    CONST robtarget T1339:=[[116.540134,72.670297,13.200015],[0.000000,0.000000,1.000000,0.000000],[0,0,-1,0],[9E+09,9E+09,9E+09,9E+09,9E+09,9E+09]];
    CONST robtarget T1340:=[[116.540134,87.329711,13.200015],[0.000000,0.000000,1.000000,0.000000],[0,0,-1,0],[9E+09,9E+09,9E+09,9E+09,9E+09,9E+09]];
    CONST robtarget T1341:=[[116.540134,114.115099,13.200015],[0.000000,0.000000,1.000000,0.000000],[0,0,-1,0],[9E+09,9E+09,9E+09,9E+09,9E+09,9E+09]];
    CONST robtarget T1342:=[[117.800139,112.721391,13.200015],[0.000000,0.000000,1.000000,0.000000],[0,0,-1,0],[9E+09,9E+09,9E+09,9E+09,9E+09,9E+09]];
    CONST robtarget T1343:=[[117.800139,86.948670,13.200015],[0.000000,0.000000,1.000000,0.000000],[0,0,-1,0],[9E+09,9E+09,9E+09,9E+09,9E+09,9E+09]];
    CONST robtarget T1344:=[[117.800139,73.051337,13.200015],[0.000000,0.000000,1.000000,0.000000],[0,0,-1,0],[9E+09,9E+09,9E+09,9E+09,9E+09,9E+09]];
    CONST robtarget T1345:=[[117.800139,47.278617,13.200015],[0.000000,0.000000,1.000000,0.000000],[0,0,-1,0],[9E+09,9E+09,9E+09,9E+09,9E+09,9E+09]];
    CONST robtarget T1346:=[[119.060143,48.787854,13.200015],[0.000000,0.000000,1.000000,0.000000],[0,0,-1,0],[9E+09,9E+09,9E+09,9E+09,9E+09,9E+09]];
    CONST robtarget T1347:=[[119.060143,73.708792,13.200015],[0.000000,0.000000,1.000000,0.000000],[0,0,-1,0],[9E+09,9E+09,9E+09,9E+09,9E+09,9E+09]];
    CONST robtarget T1348:=[[119.060143,86.291215,13.200015],[0.000000,0.000000,1.000000,0.000000],[0,0,-1,0],[9E+09,9E+09,9E+09,9E+09,9E+09,9E+09]];
    CONST robtarget T1349:=[[119.060143,111.212154,13.200015],[0.000000,0.000000,1.000000,0.000000],[0,0,-1,0],[9E+09,9E+09,9E+09,9E+09,9E+09,9E+09]];
    CONST robtarget T1350:=[[120.320148,109.560940,13.200015],[0.000000,0.000000,1.000000,0.000000],[0,0,-1,0],[9E+09,9E+09,9E+09,9E+09,9E+09,9E+09]];
    CONST robtarget T1351:=[[120.320148,85.271589,13.200015],[0.000000,0.000000,1.000000,0.000000],[0,0,-1,0],[9E+09,9E+09,9E+09,9E+09,9E+09,9E+09]];
    CONST robtarget T1352:=[[120.320148,74.728418,13.200015],[0.000000,0.000000,1.000000,0.000000],[0,0,-1,0],[9E+09,9E+09,9E+09,9E+09,9E+09,9E+09]];
    CONST robtarget T1353:=[[120.320148,50.439068,13.200015],[0.000000,0.000000,1.000000,0.000000],[0,0,-1,0],[9E+09,9E+09,9E+09,9E+09,9E+09,9E+09]];
    CONST robtarget T1354:=[[121.580152,52.240778,13.200015],[0.000000,0.000000,1.000000,0.000000],[0,0,-1,0],[9E+09,9E+09,9E+09,9E+09,9E+09,9E+09]];
    CONST robtarget T1355:=[[121.580152,76.422528,13.200015],[0.000000,0.000000,1.000000,0.000000],[0,0,-1,0],[9E+09,9E+09,9E+09,9E+09,9E+09,9E+09]];
    CONST robtarget T1356:=[[121.580152,83.577479,13.200015],[0.000000,0.000000,1.000000,0.000000],[0,0,-1,0],[9E+09,9E+09,9E+09,9E+09,9E+09,9E+09]];
    CONST robtarget T1357:=[[121.580152,107.759230,13.200015],[0.000000,0.000000,1.000000,0.000000],[0,0,-1,0],[9E+09,9E+09,9E+09,9E+09,9E+09,9E+09]];
    CONST robtarget T1358:=[[122.840157,105.775934,13.200015],[0.000000,0.000000,1.000000,0.000000],[0,0,-1,0],[9E+09,9E+09,9E+09,9E+09,9E+09,9E+09]];
    CONST robtarget T1359:=[[122.840157,54.224074,13.200015],[0.000000,0.000000,1.000000,0.000000],[0,0,-1,0],[9E+09,9E+09,9E+09,9E+09,9E+09,9E+09]];
    CONST robtarget T1360:=[[124.100161,56.444690,13.200015],[0.000000,0.000000,1.000000,0.000000],[0,0,-1,0],[9E+09,9E+09,9E+09,9E+09,9E+09,9E+09]];
    CONST robtarget T1361:=[[124.100161,103.555317,13.200015],[0.000000,0.000000,1.000000,0.000000],[0,0,-1,0],[9E+09,9E+09,9E+09,9E+09,9E+09,9E+09]];
    CONST robtarget T1362:=[[125.360166,101.007928,13.200015],[0.000000,0.000000,1.000000,0.000000],[0,0,-1,0],[9E+09,9E+09,9E+09,9E+09,9E+09,9E+09]];
    CONST robtarget T1363:=[[125.360166,58.992080,13.200015],[0.000000,0.000000,1.000000,0.000000],[0,0,-1,0],[9E+09,9E+09,9E+09,9E+09,9E+09,9E+09]];
    CONST robtarget T1364:=[[126.620170,61.953657,13.200015],[0.000000,0.000000,1.000000,0.000000],[0,0,-1,0],[9E+09,9E+09,9E+09,9E+09,9E+09,9E+09]];
    CONST robtarget T1365:=[[126.620170,98.046351,13.200015],[0.000000,0.000000,1.000000,0.000000],[0,0,-1,0],[9E+09,9E+09,9E+09,9E+09,9E+09,9E+09]];
    CONST robtarget T1366:=[[127.880175,94.360756,13.200015],[0.000000,0.000000,1.000000,0.000000],[0,0,-1,0],[9E+09,9E+09,9E+09,9E+09,9E+09,9E+09]];
    CONST robtarget T1367:=[[127.880175,65.639251,13.200015],[0.000000,0.000000,1.000000,0.000000],[0,0,-1,0],[9E+09,9E+09,9E+09,9E+09,9E+09,9E+09]];
    CONST robtarget T1368:=[[129.140179,70.797151,13.200015],[0.000000,0.000000,1.000000,0.000000],[0,0,-1,0],[9E+09,9E+09,9E+09,9E+09,9E+09,9E+09]];
    CONST robtarget T1369:=[[129.140179,89.202857,13.200015],[0.000000,0.000000,1.000000,0.000000],[0,0,-1,0],[9E+09,9E+09,9E+09,9E+09,9E+09,9E+09]];
    CONST robtarget T1370:=[[129.140179,70.797151,13.900025],[0.000000,0.000000,1.000000,0.000000],[0,0,-1,0],[9E+09,9E+09,9E+09,9E+09,9E+09,9E+09]];
    CONST robtarget T1371:=[[129.140179,89.202857,13.900025],[0.000000,0.000000,1.000000,0.000000],[0,0,-1,0],[9E+09,9E+09,9E+09,9E+09,9E+09,9E+09]];
    CONST robtarget T1372:=[[129.140179,70.797151,13.900025],[0.000000,0.000000,1.000000,0.000000],[0,0,-1,0],[9E+09,9E+09,9E+09,9E+09,9E+09,9E+09]];
    CONST robtarget T1373:=[[129.140179,89.202857,13.900025],[0.000000,0.000000,1.000000,0.000000],[0,0,-1,0],[9E+09,9E+09,9E+09,9E+09,9E+09,9E+09]];
    CONST robtarget T1374:=[[127.880175,94.360756,13.900025],[0.000000,0.000000,1.000000,0.000000],[0,0,-1,0],[9E+09,9E+09,9E+09,9E+09,9E+09,9E+09]];
    CONST robtarget T1375:=[[127.880175,65.639251,13.900025],[0.000000,0.000000,1.000000,0.000000],[0,0,-1,0],[9E+09,9E+09,9E+09,9E+09,9E+09,9E+09]];
    CONST robtarget T1376:=[[126.620170,61.953657,13.900025],[0.000000,0.000000,1.000000,0.000000],[0,0,-1,0],[9E+09,9E+09,9E+09,9E+09,9E+09,9E+09]];
    CONST robtarget T1377:=[[126.620170,98.046351,13.900025],[0.000000,0.000000,1.000000,0.000000],[0,0,-1,0],[9E+09,9E+09,9E+09,9E+09,9E+09,9E+09]];
    CONST robtarget T1378:=[[125.360166,101.007928,13.900025],[0.000000,0.000000,1.000000,0.000000],[0,0,-1,0],[9E+09,9E+09,9E+09,9E+09,9E+09,9E+09]];
    CONST robtarget T1379:=[[125.360166,58.992080,13.900025],[0.000000,0.000000,1.000000,0.000000],[0,0,-1,0],[9E+09,9E+09,9E+09,9E+09,9E+09,9E+09]];
    CONST robtarget T1380:=[[124.100161,56.444690,13.900025],[0.000000,0.000000,1.000000,0.000000],[0,0,-1,0],[9E+09,9E+09,9E+09,9E+09,9E+09,9E+09]];
    CONST robtarget T1381:=[[124.100161,103.555317,13.900025],[0.000000,0.000000,1.000000,0.000000],[0,0,-1,0],[9E+09,9E+09,9E+09,9E+09,9E+09,9E+09]];
    CONST robtarget T1382:=[[122.840157,105.775934,13.900025],[0.000000,0.000000,1.000000,0.000000],[0,0,-1,0],[9E+09,9E+09,9E+09,9E+09,9E+09,9E+09]];
    CONST robtarget T1383:=[[122.840157,54.224074,13.900025],[0.000000,0.000000,1.000000,0.000000],[0,0,-1,0],[9E+09,9E+09,9E+09,9E+09,9E+09,9E+09]];
    CONST robtarget T1384:=[[121.580152,52.240778,13.900025],[0.000000,0.000000,1.000000,0.000000],[0,0,-1,0],[9E+09,9E+09,9E+09,9E+09,9E+09,9E+09]];
    CONST robtarget T1385:=[[121.580152,76.422528,13.900025],[0.000000,0.000000,1.000000,0.000000],[0,0,-1,0],[9E+09,9E+09,9E+09,9E+09,9E+09,9E+09]];
    CONST robtarget T1386:=[[121.580152,83.577479,13.900025],[0.000000,0.000000,1.000000,0.000000],[0,0,-1,0],[9E+09,9E+09,9E+09,9E+09,9E+09,9E+09]];
    CONST robtarget T1387:=[[121.580152,107.759230,13.900025],[0.000000,0.000000,1.000000,0.000000],[0,0,-1,0],[9E+09,9E+09,9E+09,9E+09,9E+09,9E+09]];
    CONST robtarget T1388:=[[120.320148,109.560940,13.900025],[0.000000,0.000000,1.000000,0.000000],[0,0,-1,0],[9E+09,9E+09,9E+09,9E+09,9E+09,9E+09]];
    CONST robtarget T1389:=[[120.320148,85.271589,13.900025],[0.000000,0.000000,1.000000,0.000000],[0,0,-1,0],[9E+09,9E+09,9E+09,9E+09,9E+09,9E+09]];
    CONST robtarget T1390:=[[120.320148,74.728418,13.900025],[0.000000,0.000000,1.000000,0.000000],[0,0,-1,0],[9E+09,9E+09,9E+09,9E+09,9E+09,9E+09]];
    CONST robtarget T1391:=[[120.320148,50.439068,13.900025],[0.000000,0.000000,1.000000,0.000000],[0,0,-1,0],[9E+09,9E+09,9E+09,9E+09,9E+09,9E+09]];
    CONST robtarget T1392:=[[119.060143,48.787854,13.900025],[0.000000,0.000000,1.000000,0.000000],[0,0,-1,0],[9E+09,9E+09,9E+09,9E+09,9E+09,9E+09]];
    CONST robtarget T1393:=[[119.060143,73.708792,13.900025],[0.000000,0.000000,1.000000,0.000000],[0,0,-1,0],[9E+09,9E+09,9E+09,9E+09,9E+09,9E+09]];
    CONST robtarget T1394:=[[119.060143,86.291215,13.900025],[0.000000,0.000000,1.000000,0.000000],[0,0,-1,0],[9E+09,9E+09,9E+09,9E+09,9E+09,9E+09]];
    CONST robtarget T1395:=[[119.060143,111.212154,13.900025],[0.000000,0.000000,1.000000,0.000000],[0,0,-1,0],[9E+09,9E+09,9E+09,9E+09,9E+09,9E+09]];
    CONST robtarget T1396:=[[117.800139,112.721391,13.900025],[0.000000,0.000000,1.000000,0.000000],[0,0,-1,0],[9E+09,9E+09,9E+09,9E+09,9E+09,9E+09]];
    CONST robtarget T1397:=[[117.800139,86.948670,13.900025],[0.000000,0.000000,1.000000,0.000000],[0,0,-1,0],[9E+09,9E+09,9E+09,9E+09,9E+09,9E+09]];
    CONST robtarget T1398:=[[117.800139,73.051337,13.900025],[0.000000,0.000000,1.000000,0.000000],[0,0,-1,0],[9E+09,9E+09,9E+09,9E+09,9E+09,9E+09]];
    CONST robtarget T1399:=[[117.800139,47.278617,13.900025],[0.000000,0.000000,1.000000,0.000000],[0,0,-1,0],[9E+09,9E+09,9E+09,9E+09,9E+09,9E+09]];
    CONST robtarget T1400:=[[116.540134,45.884908,13.900025],[0.000000,0.000000,1.000000,0.000000],[0,0,-1,0],[9E+09,9E+09,9E+09,9E+09,9E+09,9E+09]];
    CONST robtarget T1401:=[[116.540134,72.670297,13.900025],[0.000000,0.000000,1.000000,0.000000],[0,0,-1,0],[9E+09,9E+09,9E+09,9E+09,9E+09,9E+09]];
    CONST robtarget T1402:=[[116.540134,87.329711,13.900025],[0.000000,0.000000,1.000000,0.000000],[0,0,-1,0],[9E+09,9E+09,9E+09,9E+09,9E+09,9E+09]];
    CONST robtarget T1403:=[[116.540134,114.115099,13.900025],[0.000000,0.000000,1.000000,0.000000],[0,0,-1,0],[9E+09,9E+09,9E+09,9E+09,9E+09,9E+09]];
    CONST robtarget T1404:=[[115.280130,115.412758,13.900025],[0.000000,0.000000,1.000000,0.000000],[0,0,-1,0],[9E+09,9E+09,9E+09,9E+09,9E+09,9E+09]];
    CONST robtarget T1405:=[[115.280130,87.487316,13.900025],[0.000000,0.000000,1.000000,0.000000],[0,0,-1,0],[9E+09,9E+09,9E+09,9E+09,9E+09,9E+09]];
    CONST robtarget T1406:=[[115.280130,72.512692,13.900025],[0.000000,0.000000,1.000000,0.000000],[0,0,-1,0],[9E+09,9E+09,9E+09,9E+09,9E+09,9E+09]];
    CONST robtarget T1407:=[[115.280130,44.587250,13.900025],[0.000000,0.000000,1.000000,0.000000],[0,0,-1,0],[9E+09,9E+09,9E+09,9E+09,9E+09,9E+09]];
    CONST robtarget T1408:=[[114.020125,43.373063,13.900025],[0.000000,0.000000,1.000000,0.000000],[0,0,-1,0],[9E+09,9E+09,9E+09,9E+09,9E+09,9E+09]];
    CONST robtarget T1409:=[[114.020125,72.576253,13.900025],[0.000000,0.000000,1.000000,0.000000],[0,0,-1,0],[9E+09,9E+09,9E+09,9E+09,9E+09,9E+09]];
    CONST robtarget T1410:=[[114.020125,87.423755,13.900025],[0.000000,0.000000,1.000000,0.000000],[0,0,-1,0],[9E+09,9E+09,9E+09,9E+09,9E+09,9E+09]];
    CONST robtarget T1411:=[[114.020125,116.626944,13.900025],[0.000000,0.000000,1.000000,0.000000],[0,0,-1,0],[9E+09,9E+09,9E+09,9E+09,9E+09,9E+09]];
    CONST robtarget T1412:=[[112.760121,117.767805,13.900025],[0.000000,0.000000,1.000000,0.000000],[0,0,-1,0],[9E+09,9E+09,9E+09,9E+09,9E+09,9E+09]];
    CONST robtarget T1413:=[[112.760121,87.152583,13.900025],[0.000000,0.000000,1.000000,0.000000],[0,0,-1,0],[9E+09,9E+09,9E+09,9E+09,9E+09,9E+09]];
    CONST robtarget T1414:=[[112.760121,72.847425,13.900025],[0.000000,0.000000,1.000000,0.000000],[0,0,-1,0],[9E+09,9E+09,9E+09,9E+09,9E+09,9E+09]];
    CONST robtarget T1415:=[[112.760121,42.232203,13.900025],[0.000000,0.000000,1.000000,0.000000],[0,0,-1,0],[9E+09,9E+09,9E+09,9E+09,9E+09,9E+09]];
    CONST robtarget T1416:=[[111.500116,41.180273,13.900025],[0.000000,0.000000,1.000000,0.000000],[0,0,-1,0],[9E+09,9E+09,9E+09,9E+09,9E+09,9E+09]];
    CONST robtarget T1417:=[[111.500116,73.379202,13.900025],[0.000000,0.000000,1.000000,0.000000],[0,0,-1,0],[9E+09,9E+09,9E+09,9E+09,9E+09,9E+09]];
    CONST robtarget T1418:=[[111.500116,86.620805,13.900025],[0.000000,0.000000,1.000000,0.000000],[0,0,-1,0],[9E+09,9E+09,9E+09,9E+09,9E+09,9E+09]];
    CONST robtarget T1419:=[[111.500116,118.819735,13.900025],[0.000000,0.000000,1.000000,0.000000],[0,0,-1,0],[9E+09,9E+09,9E+09,9E+09,9E+09,9E+09]];
    CONST robtarget T1420:=[[110.240112,119.803025,13.900025],[0.000000,0.000000,1.000000,0.000000],[0,0,-1,0],[9E+09,9E+09,9E+09,9E+09,9E+09,9E+09]];
    CONST robtarget T1421:=[[110.240112,85.779969,13.900025],[0.000000,0.000000,1.000000,0.000000],[0,0,-1,0],[9E+09,9E+09,9E+09,9E+09,9E+09,9E+09]];
    CONST robtarget T1422:=[[110.240112,74.220038,13.900025],[0.000000,0.000000,1.000000,0.000000],[0,0,-1,0],[9E+09,9E+09,9E+09,9E+09,9E+09,9E+09]];
    CONST robtarget T1423:=[[110.240112,40.196983,13.900025],[0.000000,0.000000,1.000000,0.000000],[0,0,-1,0],[9E+09,9E+09,9E+09,9E+09,9E+09,9E+09]];
    CONST robtarget T1424:=[[108.980107,39.265681,13.900025],[0.000000,0.000000,1.000000,0.000000],[0,0,-1,0],[9E+09,9E+09,9E+09,9E+09,9E+09,9E+09]];
    CONST robtarget T1425:=[[108.980107,75.547902,13.900025],[0.000000,0.000000,1.000000,0.000000],[0,0,-1,0],[9E+09,9E+09,9E+09,9E+09,9E+09,9E+09]];
    CONST robtarget T1426:=[[108.980107,84.452106,13.900025],[0.000000,0.000000,1.000000,0.000000],[0,0,-1,0],[9E+09,9E+09,9E+09,9E+09,9E+09,9E+09]];
    CONST robtarget T1427:=[[108.980107,120.734326,13.900025],[0.000000,0.000000,1.000000,0.000000],[0,0,-1,0],[9E+09,9E+09,9E+09,9E+09,9E+09,9E+09]];
    CONST robtarget T1428:=[[107.720103,121.607260,13.900025],[0.000000,0.000000,1.000000,0.000000],[0,0,-1,0],[9E+09,9E+09,9E+09,9E+09,9E+09,9E+09]];
    CONST robtarget T1429:=[[107.720103,81.789524,13.900025],[0.000000,0.000000,1.000000,0.000000],[0,0,-1,0],[9E+09,9E+09,9E+09,9E+09,9E+09,9E+09]];
    CONST robtarget T1430:=[[107.720103,78.210483,13.900025],[0.000000,0.000000,1.000000,0.000000],[0,0,-1,0],[9E+09,9E+09,9E+09,9E+09,9E+09,9E+09]];
    CONST robtarget T1431:=[[107.720103,38.392748,13.900025],[0.000000,0.000000,1.000000,0.000000],[0,0,-1,0],[9E+09,9E+09,9E+09,9E+09,9E+09,9E+09]];
    CONST robtarget T1432:=[[106.460098,37.589739,13.900025],[0.000000,0.000000,1.000000,0.000000],[0,0,-1,0],[9E+09,9E+09,9E+09,9E+09,9E+09,9E+09]];
    CONST robtarget T1433:=[[106.460098,122.410268,13.900025],[0.000000,0.000000,1.000000,0.000000],[0,0,-1,0],[9E+09,9E+09,9E+09,9E+09,9E+09,9E+09]];
    CONST robtarget T1434:=[[105.200094,123.174878,13.900025],[0.000000,0.000000,1.000000,0.000000],[0,0,-1,0],[9E+09,9E+09,9E+09,9E+09,9E+09,9E+09]];
    CONST robtarget T1435:=[[105.200094,36.825129,13.900025],[0.000000,0.000000,1.000000,0.000000],[0,0,-1,0],[9E+09,9E+09,9E+09,9E+09,9E+09,9E+09]];
    CONST robtarget T1436:=[[103.940089,36.110177,13.900025],[0.000000,0.000000,1.000000,0.000000],[0,0,-1,0],[9E+09,9E+09,9E+09,9E+09,9E+09,9E+09]];
    CONST robtarget T1437:=[[103.940089,123.889831,13.900025],[0.000000,0.000000,1.000000,0.000000],[0,0,-1,0],[9E+09,9E+09,9E+09,9E+09,9E+09,9E+09]];
    CONST robtarget T1438:=[[102.680085,124.546114,13.900025],[0.000000,0.000000,1.000000,0.000000],[0,0,-1,0],[9E+09,9E+09,9E+09,9E+09,9E+09,9E+09]];
    CONST robtarget T1439:=[[102.680085,35.453894,13.900025],[0.000000,0.000000,1.000000,0.000000],[0,0,-1,0],[9E+09,9E+09,9E+09,9E+09,9E+09,9E+09]];
    CONST robtarget T1440:=[[101.420080,34.827050,13.900025],[0.000000,0.000000,1.000000,0.000000],[0,0,-1,0],[9E+09,9E+09,9E+09,9E+09,9E+09,9E+09]];
    CONST robtarget T1441:=[[101.420080,125.172958,13.900025],[0.000000,0.000000,1.000000,0.000000],[0,0,-1,0],[9E+09,9E+09,9E+09,9E+09,9E+09,9E+09]];
    CONST robtarget T1442:=[[100.160076,125.745278,13.900025],[0.000000,0.000000,1.000000,0.000000],[0,0,-1,0],[9E+09,9E+09,9E+09,9E+09,9E+09,9E+09]];
    CONST robtarget T1443:=[[100.160076,34.254730,13.900025],[0.000000,0.000000,1.000000,0.000000],[0,0,-1,0],[9E+09,9E+09,9E+09,9E+09,9E+09,9E+09]];
    CONST robtarget T1444:=[[98.900071,33.722290,13.900025],[0.000000,0.000000,1.000000,0.000000],[0,0,-1,0],[9E+09,9E+09,9E+09,9E+09,9E+09,9E+09]];
    CONST robtarget T1445:=[[98.900071,126.277717,13.900025],[0.000000,0.000000,1.000000,0.000000],[0,0,-1,0],[9E+09,9E+09,9E+09,9E+09,9E+09,9E+09]];
    CONST robtarget T1446:=[[97.640067,126.783143,13.900025],[0.000000,0.000000,1.000000,0.000000],[0,0,-1,0],[9E+09,9E+09,9E+09,9E+09,9E+09,9E+09]];
    CONST robtarget T1447:=[[97.640067,33.216864,13.900025],[0.000000,0.000000,1.000000,0.000000],[0,0,-1,0],[9E+09,9E+09,9E+09,9E+09,9E+09,9E+09]];
    CONST robtarget T1448:=[[96.380062,32.772318,13.900025],[0.000000,0.000000,1.000000,0.000000],[0,0,-1,0],[9E+09,9E+09,9E+09,9E+09,9E+09,9E+09]];
    CONST robtarget T1449:=[[96.380062,127.227690,13.900025],[0.000000,0.000000,1.000000,0.000000],[0,0,-1,0],[9E+09,9E+09,9E+09,9E+09,9E+09,9E+09]];
    CONST robtarget T1450:=[[95.120058,127.652167,13.900025],[0.000000,0.000000,1.000000,0.000000],[0,0,-1,0],[9E+09,9E+09,9E+09,9E+09,9E+09,9E+09]];
    CONST robtarget T1451:=[[95.120058,32.347841,13.900025],[0.000000,0.000000,1.000000,0.000000],[0,0,-1,0],[9E+09,9E+09,9E+09,9E+09,9E+09,9E+09]];
    CONST robtarget T1452:=[[93.860053,31.969479,13.900025],[0.000000,0.000000,1.000000,0.000000],[0,0,-1,0],[9E+09,9E+09,9E+09,9E+09,9E+09,9E+09]];
    CONST robtarget T1453:=[[93.860053,128.030529,13.900025],[0.000000,0.000000,1.000000,0.000000],[0,0,-1,0],[9E+09,9E+09,9E+09,9E+09,9E+09,9E+09]];
    CONST robtarget T1454:=[[92.600049,128.374988,13.900025],[0.000000,0.000000,1.000000,0.000000],[0,0,-1,0],[9E+09,9E+09,9E+09,9E+09,9E+09,9E+09]];
    CONST robtarget T1455:=[[92.600049,31.625019,13.900025],[0.000000,0.000000,1.000000,0.000000],[0,0,-1,0],[9E+09,9E+09,9E+09,9E+09,9E+09,9E+09]];
    CONST robtarget T1456:=[[91.340044,31.307526,13.900025],[0.000000,0.000000,1.000000,0.000000],[0,0,-1,0],[9E+09,9E+09,9E+09,9E+09,9E+09,9E+09]];
    CONST robtarget T1457:=[[91.340044,128.692481,13.900025],[0.000000,0.000000,1.000000,0.000000],[0,0,-1,0],[9E+09,9E+09,9E+09,9E+09,9E+09,9E+09]];
    CONST robtarget T1458:=[[90.080040,128.960575,13.900025],[0.000000,0.000000,1.000000,0.000000],[0,0,-1,0],[9E+09,9E+09,9E+09,9E+09,9E+09,9E+09]];
    CONST robtarget T1459:=[[90.080040,31.039433,13.900025],[0.000000,0.000000,1.000000,0.000000],[0,0,-1,0],[9E+09,9E+09,9E+09,9E+09,9E+09,9E+09]];
    CONST robtarget T1460:=[[88.820035,30.786444,13.900025],[0.000000,0.000000,1.000000,0.000000],[0,0,-1,0],[9E+09,9E+09,9E+09,9E+09,9E+09,9E+09]];
    CONST robtarget T1461:=[[88.820035,129.213563,13.900025],[0.000000,0.000000,1.000000,0.000000],[0,0,-1,0],[9E+09,9E+09,9E+09,9E+09,9E+09,9E+09]];
    CONST robtarget T1462:=[[87.560031,129.413129,13.900025],[0.000000,0.000000,1.000000,0.000000],[0,0,-1,0],[9E+09,9E+09,9E+09,9E+09,9E+09,9E+09]];
    CONST robtarget T1463:=[[87.560031,30.586879,13.900025],[0.000000,0.000000,1.000000,0.000000],[0,0,-1,0],[9E+09,9E+09,9E+09,9E+09,9E+09,9E+09]];
    CONST robtarget T1464:=[[86.300026,30.406130,13.900025],[0.000000,0.000000,1.000000,0.000000],[0,0,-1,0],[9E+09,9E+09,9E+09,9E+09,9E+09,9E+09]];
    CONST robtarget T1465:=[[86.300026,40.937335,13.900025],[0.000000,0.000000,1.000000,0.000000],[0,0,-1,0],[9E+09,9E+09,9E+09,9E+09,9E+09,9E+09]];
    CONST robtarget T1466:=[[86.300026,49.062665,13.900025],[0.000000,0.000000,1.000000,0.000000],[0,0,-1,0],[9E+09,9E+09,9E+09,9E+09,9E+09,9E+09]];
    CONST robtarget T1467:=[[86.300026,75.937339,13.900025],[0.000000,0.000000,1.000000,0.000000],[0,0,-1,0],[9E+09,9E+09,9E+09,9E+09,9E+09,9E+09]];
    CONST robtarget T1468:=[[86.300026,84.062668,13.900025],[0.000000,0.000000,1.000000,0.000000],[0,0,-1,0],[9E+09,9E+09,9E+09,9E+09,9E+09,9E+09]];
    CONST robtarget T1469:=[[86.300026,110.937342,13.900025],[0.000000,0.000000,1.000000,0.000000],[0,0,-1,0],[9E+09,9E+09,9E+09,9E+09,9E+09,9E+09]];
    CONST robtarget T1470:=[[86.300026,119.062672,13.900025],[0.000000,0.000000,1.000000,0.000000],[0,0,-1,0],[9E+09,9E+09,9E+09,9E+09,9E+09,9E+09]];
    CONST robtarget T1471:=[[86.300026,129.593877,13.900025],[0.000000,0.000000,1.000000,0.000000],[0,0,-1,0],[9E+09,9E+09,9E+09,9E+09,9E+09,9E+09]];
    CONST robtarget T1472:=[[85.040022,129.735844,13.900025],[0.000000,0.000000,1.000000,0.000000],[0,0,-1,0],[9E+09,9E+09,9E+09,9E+09,9E+09,9E+09]];
    CONST robtarget T1473:=[[85.040022,120.544921,13.900025],[0.000000,0.000000,1.000000,0.000000],[0,0,-1,0],[9E+09,9E+09,9E+09,9E+09,9E+09,9E+09]];
    CONST robtarget T1474:=[[85.040022,109.455091,13.900025],[0.000000,0.000000,1.000000,0.000000],[0,0,-1,0],[9E+09,9E+09,9E+09,9E+09,9E+09,9E+09]];
    CONST robtarget T1475:=[[85.040022,85.544918,13.900025],[0.000000,0.000000,1.000000,0.000000],[0,0,-1,0],[9E+09,9E+09,9E+09,9E+09,9E+09,9E+09]];
    CONST robtarget T1476:=[[85.040022,74.455090,13.900025],[0.000000,0.000000,1.000000,0.000000],[0,0,-1,0],[9E+09,9E+09,9E+09,9E+09,9E+09,9E+09]];
    CONST robtarget T1477:=[[85.040022,50.544916,13.900025],[0.000000,0.000000,1.000000,0.000000],[0,0,-1,0],[9E+09,9E+09,9E+09,9E+09,9E+09,9E+09]];
    CONST robtarget T1478:=[[85.040022,39.455086,13.900025],[0.000000,0.000000,1.000000,0.000000],[0,0,-1,0],[9E+09,9E+09,9E+09,9E+09,9E+09,9E+09]];
    CONST robtarget T1479:=[[85.040022,30.264163,13.900025],[0.000000,0.000000,1.000000,0.000000],[0,0,-1,0],[9E+09,9E+09,9E+09,9E+09,9E+09,9E+09]];
    CONST robtarget T1480:=[[83.780017,30.153959,13.900025],[0.000000,0.000000,1.000000,0.000000],[0,0,-1,0],[9E+09,9E+09,9E+09,9E+09,9E+09,9E+09]];
    CONST robtarget T1481:=[[83.780017,38.524551,13.900025],[0.000000,0.000000,1.000000,0.000000],[0,0,-1,0],[9E+09,9E+09,9E+09,9E+09,9E+09,9E+09]];
    CONST robtarget T1482:=[[83.780017,51.475451,13.900025],[0.000000,0.000000,1.000000,0.000000],[0,0,-1,0],[9E+09,9E+09,9E+09,9E+09,9E+09,9E+09]];
    CONST robtarget T1483:=[[83.780017,73.524553,13.900025],[0.000000,0.000000,1.000000,0.000000],[0,0,-1,0],[9E+09,9E+09,9E+09,9E+09,9E+09,9E+09]];
    CONST robtarget T1484:=[[83.780017,86.475455,13.900025],[0.000000,0.000000,1.000000,0.000000],[0,0,-1,0],[9E+09,9E+09,9E+09,9E+09,9E+09,9E+09]];
    CONST robtarget T1485:=[[83.780017,108.524556,13.900025],[0.000000,0.000000,1.000000,0.000000],[0,0,-1,0],[9E+09,9E+09,9E+09,9E+09,9E+09,9E+09]];
    CONST robtarget T1486:=[[83.780017,121.475457,13.900025],[0.000000,0.000000,1.000000,0.000000],[0,0,-1,0],[9E+09,9E+09,9E+09,9E+09,9E+09,9E+09]];
    CONST robtarget T1487:=[[83.780017,129.846049,13.900025],[0.000000,0.000000,1.000000,0.000000],[0,0,-1,0],[9E+09,9E+09,9E+09,9E+09,9E+09,9E+09]];
    CONST robtarget T1488:=[[82.520013,129.931001,13.900025],[0.000000,0.000000,1.000000,0.000000],[0,0,-1,0],[9E+09,9E+09,9E+09,9E+09,9E+09,9E+09]];
    CONST robtarget T1489:=[[82.520013,122.050628,13.900025],[0.000000,0.000000,1.000000,0.000000],[0,0,-1,0],[9E+09,9E+09,9E+09,9E+09,9E+09,9E+09]];
    CONST robtarget T1490:=[[82.520013,107.949384,13.900025],[0.000000,0.000000,1.000000,0.000000],[0,0,-1,0],[9E+09,9E+09,9E+09,9E+09,9E+09,9E+09]];
    CONST robtarget T1491:=[[82.520013,87.050626,13.900025],[0.000000,0.000000,1.000000,0.000000],[0,0,-1,0],[9E+09,9E+09,9E+09,9E+09,9E+09,9E+09]];
    CONST robtarget T1492:=[[82.520013,72.949381,13.900025],[0.000000,0.000000,1.000000,0.000000],[0,0,-1,0],[9E+09,9E+09,9E+09,9E+09,9E+09,9E+09]];
    CONST robtarget T1493:=[[82.520013,52.050624,13.900025],[0.000000,0.000000,1.000000,0.000000],[0,0,-1,0],[9E+09,9E+09,9E+09,9E+09,9E+09,9E+09]];
    CONST robtarget T1494:=[[82.520013,37.949379,13.900025],[0.000000,0.000000,1.000000,0.000000],[0,0,-1,0],[9E+09,9E+09,9E+09,9E+09,9E+09,9E+09]];
    CONST robtarget T1495:=[[82.520013,30.069007,13.900025],[0.000000,0.000000,1.000000,0.000000],[0,0,-1,0],[9E+09,9E+09,9E+09,9E+09,9E+09,9E+09]];
    CONST robtarget T1496:=[[81.260008,30.028279,13.900025],[0.000000,0.000000,1.000000,0.000000],[0,0,-1,0],[9E+09,9E+09,9E+09,9E+09,9E+09,9E+09]];
    CONST robtarget T1497:=[[81.260008,37.608991,13.900025],[0.000000,0.000000,1.000000,0.000000],[0,0,-1,0],[9E+09,9E+09,9E+09,9E+09,9E+09,9E+09]];
    CONST robtarget T1498:=[[81.260008,52.391011,13.900025],[0.000000,0.000000,1.000000,0.000000],[0,0,-1,0],[9E+09,9E+09,9E+09,9E+09,9E+09,9E+09]];
    CONST robtarget T1499:=[[81.260008,72.608994,13.900025],[0.000000,0.000000,1.000000,0.000000],[0,0,-1,0],[9E+09,9E+09,9E+09,9E+09,9E+09,9E+09]];
    CONST robtarget T1500:=[[81.260008,87.391014,13.900025],[0.000000,0.000000,1.000000,0.000000],[0,0,-1,0],[9E+09,9E+09,9E+09,9E+09,9E+09,9E+09]];
    CONST robtarget T1501:=[[81.260008,107.608996,13.900025],[0.000000,0.000000,1.000000,0.000000],[0,0,-1,0],[9E+09,9E+09,9E+09,9E+09,9E+09,9E+09]];
    CONST robtarget T1502:=[[81.260008,122.391017,13.900025],[0.000000,0.000000,1.000000,0.000000],[0,0,-1,0],[9E+09,9E+09,9E+09,9E+09,9E+09,9E+09]];
    CONST robtarget T1503:=[[81.260008,129.971729,13.900025],[0.000000,0.000000,1.000000,0.000000],[0,0,-1,0],[9E+09,9E+09,9E+09,9E+09,9E+09,9E+09]];
    CONST robtarget T1504:=[[80.000004,130.000008,13.900025],[0.000000,0.000000,1.000000,0.000000],[0,0,-1,0],[9E+09,9E+09,9E+09,9E+09,9E+09,9E+09]];
    CONST robtarget T1505:=[[80.000004,122.487319,13.900025],[0.000000,0.000000,1.000000,0.000000],[0,0,-1,0],[9E+09,9E+09,9E+09,9E+09,9E+09,9E+09]];
    CONST robtarget T1506:=[[80.000004,107.512696,13.900025],[0.000000,0.000000,1.000000,0.000000],[0,0,-1,0],[9E+09,9E+09,9E+09,9E+09,9E+09,9E+09]];
    CONST robtarget T1507:=[[80.000004,87.487316,13.900025],[0.000000,0.000000,1.000000,0.000000],[0,0,-1,0],[9E+09,9E+09,9E+09,9E+09,9E+09,9E+09]];
    CONST robtarget T1508:=[[80.000004,72.512692,13.900025],[0.000000,0.000000,1.000000,0.000000],[0,0,-1,0],[9E+09,9E+09,9E+09,9E+09,9E+09,9E+09]];
    CONST robtarget T1509:=[[80.000004,52.487312,13.900025],[0.000000,0.000000,1.000000,0.000000],[0,0,-1,0],[9E+09,9E+09,9E+09,9E+09,9E+09,9E+09]];
    CONST robtarget T1510:=[[80.000004,37.512688,13.900025],[0.000000,0.000000,1.000000,0.000000],[0,0,-1,0],[9E+09,9E+09,9E+09,9E+09,9E+09,9E+09]];
    CONST robtarget T1511:=[[80.000004,30.000000,13.900025],[0.000000,0.000000,1.000000,0.000000],[0,0,-1,0],[9E+09,9E+09,9E+09,9E+09,9E+09,9E+09]];
    CONST robtarget T1512:=[[78.739999,30.028279,13.900025],[0.000000,0.000000,1.000000,0.000000],[0,0,-1,0],[9E+09,9E+09,9E+09,9E+09,9E+09,9E+09]];
    CONST robtarget T1513:=[[78.739999,37.608991,13.900025],[0.000000,0.000000,1.000000,0.000000],[0,0,-1,0],[9E+09,9E+09,9E+09,9E+09,9E+09,9E+09]];
    CONST robtarget T1514:=[[78.739999,52.391011,13.900025],[0.000000,0.000000,1.000000,0.000000],[0,0,-1,0],[9E+09,9E+09,9E+09,9E+09,9E+09,9E+09]];
    CONST robtarget T1515:=[[78.739999,72.608994,13.900025],[0.000000,0.000000,1.000000,0.000000],[0,0,-1,0],[9E+09,9E+09,9E+09,9E+09,9E+09,9E+09]];
    CONST robtarget T1516:=[[78.739999,87.391014,13.900025],[0.000000,0.000000,1.000000,0.000000],[0,0,-1,0],[9E+09,9E+09,9E+09,9E+09,9E+09,9E+09]];
    CONST robtarget T1517:=[[78.739999,107.608996,13.900025],[0.000000,0.000000,1.000000,0.000000],[0,0,-1,0],[9E+09,9E+09,9E+09,9E+09,9E+09,9E+09]];
    CONST robtarget T1518:=[[78.739999,122.391017,13.900025],[0.000000,0.000000,1.000000,0.000000],[0,0,-1,0],[9E+09,9E+09,9E+09,9E+09,9E+09,9E+09]];
    CONST robtarget T1519:=[[78.739999,129.971729,13.900025],[0.000000,0.000000,1.000000,0.000000],[0,0,-1,0],[9E+09,9E+09,9E+09,9E+09,9E+09,9E+09]];
    CONST robtarget T1520:=[[77.479995,129.931001,13.900025],[0.000000,0.000000,1.000000,0.000000],[0,0,-1,0],[9E+09,9E+09,9E+09,9E+09,9E+09,9E+09]];
    CONST robtarget T1521:=[[77.479995,122.050628,13.900025],[0.000000,0.000000,1.000000,0.000000],[0,0,-1,0],[9E+09,9E+09,9E+09,9E+09,9E+09,9E+09]];
    CONST robtarget T1522:=[[77.479995,107.949384,13.900025],[0.000000,0.000000,1.000000,0.000000],[0,0,-1,0],[9E+09,9E+09,9E+09,9E+09,9E+09,9E+09]];
    CONST robtarget T1523:=[[77.479995,87.050626,13.900025],[0.000000,0.000000,1.000000,0.000000],[0,0,-1,0],[9E+09,9E+09,9E+09,9E+09,9E+09,9E+09]];
    CONST robtarget T1524:=[[77.479995,72.949381,13.900025],[0.000000,0.000000,1.000000,0.000000],[0,0,-1,0],[9E+09,9E+09,9E+09,9E+09,9E+09,9E+09]];
    CONST robtarget T1525:=[[77.479995,52.050624,13.900025],[0.000000,0.000000,1.000000,0.000000],[0,0,-1,0],[9E+09,9E+09,9E+09,9E+09,9E+09,9E+09]];
    CONST robtarget T1526:=[[77.479995,37.949379,13.900025],[0.000000,0.000000,1.000000,0.000000],[0,0,-1,0],[9E+09,9E+09,9E+09,9E+09,9E+09,9E+09]];
    CONST robtarget T1527:=[[77.479995,30.069007,13.900025],[0.000000,0.000000,1.000000,0.000000],[0,0,-1,0],[9E+09,9E+09,9E+09,9E+09,9E+09,9E+09]];
    CONST robtarget T1528:=[[76.219990,30.153959,13.900025],[0.000000,0.000000,1.000000,0.000000],[0,0,-1,0],[9E+09,9E+09,9E+09,9E+09,9E+09,9E+09]];
    CONST robtarget T1529:=[[76.219990,38.524551,13.900025],[0.000000,0.000000,1.000000,0.000000],[0,0,-1,0],[9E+09,9E+09,9E+09,9E+09,9E+09,9E+09]];
    CONST robtarget T1530:=[[76.219990,51.475451,13.900025],[0.000000,0.000000,1.000000,0.000000],[0,0,-1,0],[9E+09,9E+09,9E+09,9E+09,9E+09,9E+09]];
    CONST robtarget T1531:=[[76.219990,73.524553,13.900025],[0.000000,0.000000,1.000000,0.000000],[0,0,-1,0],[9E+09,9E+09,9E+09,9E+09,9E+09,9E+09]];
    CONST robtarget T1532:=[[76.219990,86.475455,13.900025],[0.000000,0.000000,1.000000,0.000000],[0,0,-1,0],[9E+09,9E+09,9E+09,9E+09,9E+09,9E+09]];
    CONST robtarget T1533:=[[76.219990,108.524556,13.900025],[0.000000,0.000000,1.000000,0.000000],[0,0,-1,0],[9E+09,9E+09,9E+09,9E+09,9E+09,9E+09]];
    CONST robtarget T1534:=[[76.219990,121.475457,13.900025],[0.000000,0.000000,1.000000,0.000000],[0,0,-1,0],[9E+09,9E+09,9E+09,9E+09,9E+09,9E+09]];
    CONST robtarget T1535:=[[76.219990,129.846049,13.900025],[0.000000,0.000000,1.000000,0.000000],[0,0,-1,0],[9E+09,9E+09,9E+09,9E+09,9E+09,9E+09]];
    CONST robtarget T1536:=[[74.959986,129.735844,13.900025],[0.000000,0.000000,1.000000,0.000000],[0,0,-1,0],[9E+09,9E+09,9E+09,9E+09,9E+09,9E+09]];
    CONST robtarget T1537:=[[74.959986,120.544921,13.900025],[0.000000,0.000000,1.000000,0.000000],[0,0,-1,0],[9E+09,9E+09,9E+09,9E+09,9E+09,9E+09]];
    CONST robtarget T1538:=[[74.959986,109.455091,13.900025],[0.000000,0.000000,1.000000,0.000000],[0,0,-1,0],[9E+09,9E+09,9E+09,9E+09,9E+09,9E+09]];
    CONST robtarget T1539:=[[74.959986,85.544918,13.900025],[0.000000,0.000000,1.000000,0.000000],[0,0,-1,0],[9E+09,9E+09,9E+09,9E+09,9E+09,9E+09]];
    CONST robtarget T1540:=[[74.959986,74.455090,13.900025],[0.000000,0.000000,1.000000,0.000000],[0,0,-1,0],[9E+09,9E+09,9E+09,9E+09,9E+09,9E+09]];
    CONST robtarget T1541:=[[74.959986,50.544916,13.900025],[0.000000,0.000000,1.000000,0.000000],[0,0,-1,0],[9E+09,9E+09,9E+09,9E+09,9E+09,9E+09]];
    CONST robtarget T1542:=[[74.959986,39.455086,13.900025],[0.000000,0.000000,1.000000,0.000000],[0,0,-1,0],[9E+09,9E+09,9E+09,9E+09,9E+09,9E+09]];
    CONST robtarget T1543:=[[74.959986,30.264163,13.900025],[0.000000,0.000000,1.000000,0.000000],[0,0,-1,0],[9E+09,9E+09,9E+09,9E+09,9E+09,9E+09]];
    CONST robtarget T1544:=[[73.699981,30.406130,13.900025],[0.000000,0.000000,1.000000,0.000000],[0,0,-1,0],[9E+09,9E+09,9E+09,9E+09,9E+09,9E+09]];
    CONST robtarget T1545:=[[73.699981,40.937335,13.900025],[0.000000,0.000000,1.000000,0.000000],[0,0,-1,0],[9E+09,9E+09,9E+09,9E+09,9E+09,9E+09]];
    CONST robtarget T1546:=[[73.699981,49.062665,13.900025],[0.000000,0.000000,1.000000,0.000000],[0,0,-1,0],[9E+09,9E+09,9E+09,9E+09,9E+09,9E+09]];
    CONST robtarget T1547:=[[73.699981,75.937339,13.900025],[0.000000,0.000000,1.000000,0.000000],[0,0,-1,0],[9E+09,9E+09,9E+09,9E+09,9E+09,9E+09]];
    CONST robtarget T1548:=[[73.699981,84.062668,13.900025],[0.000000,0.000000,1.000000,0.000000],[0,0,-1,0],[9E+09,9E+09,9E+09,9E+09,9E+09,9E+09]];
    CONST robtarget T1549:=[[73.699981,110.937342,13.900025],[0.000000,0.000000,1.000000,0.000000],[0,0,-1,0],[9E+09,9E+09,9E+09,9E+09,9E+09,9E+09]];
    CONST robtarget T1550:=[[73.699981,119.062672,13.900025],[0.000000,0.000000,1.000000,0.000000],[0,0,-1,0],[9E+09,9E+09,9E+09,9E+09,9E+09,9E+09]];
    CONST robtarget T1551:=[[73.699981,129.593877,13.900025],[0.000000,0.000000,1.000000,0.000000],[0,0,-1,0],[9E+09,9E+09,9E+09,9E+09,9E+09,9E+09]];
    CONST robtarget T1552:=[[72.439977,129.413129,13.900025],[0.000000,0.000000,1.000000,0.000000],[0,0,-1,0],[9E+09,9E+09,9E+09,9E+09,9E+09,9E+09]];
    CONST robtarget T1553:=[[72.439977,30.586879,13.900025],[0.000000,0.000000,1.000000,0.000000],[0,0,-1,0],[9E+09,9E+09,9E+09,9E+09,9E+09,9E+09]];
    CONST robtarget T1554:=[[71.179972,30.786444,13.900025],[0.000000,0.000000,1.000000,0.000000],[0,0,-1,0],[9E+09,9E+09,9E+09,9E+09,9E+09,9E+09]];
    CONST robtarget T1555:=[[71.179972,129.213563,13.900025],[0.000000,0.000000,1.000000,0.000000],[0,0,-1,0],[9E+09,9E+09,9E+09,9E+09,9E+09,9E+09]];
    CONST robtarget T1556:=[[69.919968,128.960575,13.900025],[0.000000,0.000000,1.000000,0.000000],[0,0,-1,0],[9E+09,9E+09,9E+09,9E+09,9E+09,9E+09]];
    CONST robtarget T1557:=[[69.919968,31.039433,13.900025],[0.000000,0.000000,1.000000,0.000000],[0,0,-1,0],[9E+09,9E+09,9E+09,9E+09,9E+09,9E+09]];
    CONST robtarget T1558:=[[68.659963,31.307526,13.900025],[0.000000,0.000000,1.000000,0.000000],[0,0,-1,0],[9E+09,9E+09,9E+09,9E+09,9E+09,9E+09]];
    CONST robtarget T1559:=[[68.659963,128.692481,13.900025],[0.000000,0.000000,1.000000,0.000000],[0,0,-1,0],[9E+09,9E+09,9E+09,9E+09,9E+09,9E+09]];
    CONST robtarget T1560:=[[67.399959,128.374988,13.900025],[0.000000,0.000000,1.000000,0.000000],[0,0,-1,0],[9E+09,9E+09,9E+09,9E+09,9E+09,9E+09]];
    CONST robtarget T1561:=[[67.399959,31.625019,13.900025],[0.000000,0.000000,1.000000,0.000000],[0,0,-1,0],[9E+09,9E+09,9E+09,9E+09,9E+09,9E+09]];
    CONST robtarget T1562:=[[66.139954,31.969479,13.900025],[0.000000,0.000000,1.000000,0.000000],[0,0,-1,0],[9E+09,9E+09,9E+09,9E+09,9E+09,9E+09]];
    CONST robtarget T1563:=[[66.139954,128.030529,13.900025],[0.000000,0.000000,1.000000,0.000000],[0,0,-1,0],[9E+09,9E+09,9E+09,9E+09,9E+09,9E+09]];
    CONST robtarget T1564:=[[64.879950,127.652167,13.900025],[0.000000,0.000000,1.000000,0.000000],[0,0,-1,0],[9E+09,9E+09,9E+09,9E+09,9E+09,9E+09]];
    CONST robtarget T1565:=[[64.879950,32.347841,13.900025],[0.000000,0.000000,1.000000,0.000000],[0,0,-1,0],[9E+09,9E+09,9E+09,9E+09,9E+09,9E+09]];
    CONST robtarget T1566:=[[63.619945,32.772318,13.900025],[0.000000,0.000000,1.000000,0.000000],[0,0,-1,0],[9E+09,9E+09,9E+09,9E+09,9E+09,9E+09]];
    CONST robtarget T1567:=[[63.619945,127.227690,13.900025],[0.000000,0.000000,1.000000,0.000000],[0,0,-1,0],[9E+09,9E+09,9E+09,9E+09,9E+09,9E+09]];
    CONST robtarget T1568:=[[62.359941,126.783143,13.900025],[0.000000,0.000000,1.000000,0.000000],[0,0,-1,0],[9E+09,9E+09,9E+09,9E+09,9E+09,9E+09]];
    CONST robtarget T1569:=[[62.359941,33.216864,13.900025],[0.000000,0.000000,1.000000,0.000000],[0,0,-1,0],[9E+09,9E+09,9E+09,9E+09,9E+09,9E+09]];
    CONST robtarget T1570:=[[61.099936,33.722290,13.900025],[0.000000,0.000000,1.000000,0.000000],[0,0,-1,0],[9E+09,9E+09,9E+09,9E+09,9E+09,9E+09]];
    CONST robtarget T1571:=[[61.099936,126.277717,13.900025],[0.000000,0.000000,1.000000,0.000000],[0,0,-1,0],[9E+09,9E+09,9E+09,9E+09,9E+09,9E+09]];
    CONST robtarget T1572:=[[59.839932,125.745278,13.900025],[0.000000,0.000000,1.000000,0.000000],[0,0,-1,0],[9E+09,9E+09,9E+09,9E+09,9E+09,9E+09]];
    CONST robtarget T1573:=[[59.839932,34.254730,13.900025],[0.000000,0.000000,1.000000,0.000000],[0,0,-1,0],[9E+09,9E+09,9E+09,9E+09,9E+09,9E+09]];
    CONST robtarget T1574:=[[58.579927,34.827050,13.900025],[0.000000,0.000000,1.000000,0.000000],[0,0,-1,0],[9E+09,9E+09,9E+09,9E+09,9E+09,9E+09]];
    CONST robtarget T1575:=[[58.579927,125.172958,13.900025],[0.000000,0.000000,1.000000,0.000000],[0,0,-1,0],[9E+09,9E+09,9E+09,9E+09,9E+09,9E+09]];
    CONST robtarget T1576:=[[57.319923,124.546114,13.900025],[0.000000,0.000000,1.000000,0.000000],[0,0,-1,0],[9E+09,9E+09,9E+09,9E+09,9E+09,9E+09]];
    CONST robtarget T1577:=[[57.319923,35.453894,13.900025],[0.000000,0.000000,1.000000,0.000000],[0,0,-1,0],[9E+09,9E+09,9E+09,9E+09,9E+09,9E+09]];
    CONST robtarget T1578:=[[56.059918,36.110177,13.900025],[0.000000,0.000000,1.000000,0.000000],[0,0,-1,0],[9E+09,9E+09,9E+09,9E+09,9E+09,9E+09]];
    CONST robtarget T1579:=[[56.059918,123.889831,13.900025],[0.000000,0.000000,1.000000,0.000000],[0,0,-1,0],[9E+09,9E+09,9E+09,9E+09,9E+09,9E+09]];
    CONST robtarget T1580:=[[54.799914,123.174878,13.900025],[0.000000,0.000000,1.000000,0.000000],[0,0,-1,0],[9E+09,9E+09,9E+09,9E+09,9E+09,9E+09]];
    CONST robtarget T1581:=[[54.799914,36.825129,13.900025],[0.000000,0.000000,1.000000,0.000000],[0,0,-1,0],[9E+09,9E+09,9E+09,9E+09,9E+09,9E+09]];
    CONST robtarget T1582:=[[53.539909,37.589739,13.900025],[0.000000,0.000000,1.000000,0.000000],[0,0,-1,0],[9E+09,9E+09,9E+09,9E+09,9E+09,9E+09]];
    CONST robtarget T1583:=[[53.539909,122.410268,13.900025],[0.000000,0.000000,1.000000,0.000000],[0,0,-1,0],[9E+09,9E+09,9E+09,9E+09,9E+09,9E+09]];
    CONST robtarget T1584:=[[52.279905,121.607260,13.900025],[0.000000,0.000000,1.000000,0.000000],[0,0,-1,0],[9E+09,9E+09,9E+09,9E+09,9E+09,9E+09]];
    CONST robtarget T1585:=[[52.279905,81.789524,13.900025],[0.000000,0.000000,1.000000,0.000000],[0,0,-1,0],[9E+09,9E+09,9E+09,9E+09,9E+09,9E+09]];
    CONST robtarget T1586:=[[52.279905,78.210483,13.900025],[0.000000,0.000000,1.000000,0.000000],[0,0,-1,0],[9E+09,9E+09,9E+09,9E+09,9E+09,9E+09]];
    CONST robtarget T1587:=[[52.279905,38.392748,13.900025],[0.000000,0.000000,1.000000,0.000000],[0,0,-1,0],[9E+09,9E+09,9E+09,9E+09,9E+09,9E+09]];
    CONST robtarget T1588:=[[51.019900,39.265681,13.900025],[0.000000,0.000000,1.000000,0.000000],[0,0,-1,0],[9E+09,9E+09,9E+09,9E+09,9E+09,9E+09]];
    CONST robtarget T1589:=[[51.019900,75.547902,13.900025],[0.000000,0.000000,1.000000,0.000000],[0,0,-1,0],[9E+09,9E+09,9E+09,9E+09,9E+09,9E+09]];
    CONST robtarget T1590:=[[51.019900,84.452106,13.900025],[0.000000,0.000000,1.000000,0.000000],[0,0,-1,0],[9E+09,9E+09,9E+09,9E+09,9E+09,9E+09]];
    CONST robtarget T1591:=[[51.019900,120.734326,13.900025],[0.000000,0.000000,1.000000,0.000000],[0,0,-1,0],[9E+09,9E+09,9E+09,9E+09,9E+09,9E+09]];
    CONST robtarget T1592:=[[49.759896,119.803025,13.900025],[0.000000,0.000000,1.000000,0.000000],[0,0,-1,0],[9E+09,9E+09,9E+09,9E+09,9E+09,9E+09]];
    CONST robtarget T1593:=[[49.759896,85.779969,13.900025],[0.000000,0.000000,1.000000,0.000000],[0,0,-1,0],[9E+09,9E+09,9E+09,9E+09,9E+09,9E+09]];
    CONST robtarget T1594:=[[49.759896,74.220038,13.900025],[0.000000,0.000000,1.000000,0.000000],[0,0,-1,0],[9E+09,9E+09,9E+09,9E+09,9E+09,9E+09]];
    CONST robtarget T1595:=[[49.759896,40.196983,13.900025],[0.000000,0.000000,1.000000,0.000000],[0,0,-1,0],[9E+09,9E+09,9E+09,9E+09,9E+09,9E+09]];
    CONST robtarget T1596:=[[48.499891,41.180273,13.900025],[0.000000,0.000000,1.000000,0.000000],[0,0,-1,0],[9E+09,9E+09,9E+09,9E+09,9E+09,9E+09]];
    CONST robtarget T1597:=[[48.499891,73.379202,13.900025],[0.000000,0.000000,1.000000,0.000000],[0,0,-1,0],[9E+09,9E+09,9E+09,9E+09,9E+09,9E+09]];
    CONST robtarget T1598:=[[48.499891,86.620805,13.900025],[0.000000,0.000000,1.000000,0.000000],[0,0,-1,0],[9E+09,9E+09,9E+09,9E+09,9E+09,9E+09]];
    CONST robtarget T1599:=[[48.499891,118.819735,13.900025],[0.000000,0.000000,1.000000,0.000000],[0,0,-1,0],[9E+09,9E+09,9E+09,9E+09,9E+09,9E+09]];
    CONST robtarget T1600:=[[47.239887,117.767805,13.900025],[0.000000,0.000000,1.000000,0.000000],[0,0,-1,0],[9E+09,9E+09,9E+09,9E+09,9E+09,9E+09]];
    CONST robtarget T1601:=[[47.239887,87.152583,13.900025],[0.000000,0.000000,1.000000,0.000000],[0,0,-1,0],[9E+09,9E+09,9E+09,9E+09,9E+09,9E+09]];
    CONST robtarget T1602:=[[47.239887,72.847425,13.900025],[0.000000,0.000000,1.000000,0.000000],[0,0,-1,0],[9E+09,9E+09,9E+09,9E+09,9E+09,9E+09]];
    CONST robtarget T1603:=[[47.239887,42.232203,13.900025],[0.000000,0.000000,1.000000,0.000000],[0,0,-1,0],[9E+09,9E+09,9E+09,9E+09,9E+09,9E+09]];
    CONST robtarget T1604:=[[45.979882,43.373063,13.900025],[0.000000,0.000000,1.000000,0.000000],[0,0,-1,0],[9E+09,9E+09,9E+09,9E+09,9E+09,9E+09]];
    CONST robtarget T1605:=[[45.979882,72.576253,13.900025],[0.000000,0.000000,1.000000,0.000000],[0,0,-1,0],[9E+09,9E+09,9E+09,9E+09,9E+09,9E+09]];
    CONST robtarget T1606:=[[45.979882,87.423755,13.900025],[0.000000,0.000000,1.000000,0.000000],[0,0,-1,0],[9E+09,9E+09,9E+09,9E+09,9E+09,9E+09]];
    CONST robtarget T1607:=[[45.979882,116.626944,13.900025],[0.000000,0.000000,1.000000,0.000000],[0,0,-1,0],[9E+09,9E+09,9E+09,9E+09,9E+09,9E+09]];
    CONST robtarget T1608:=[[44.719878,115.412758,13.900025],[0.000000,0.000000,1.000000,0.000000],[0,0,-1,0],[9E+09,9E+09,9E+09,9E+09,9E+09,9E+09]];
    CONST robtarget T1609:=[[44.719878,87.487316,13.900025],[0.000000,0.000000,1.000000,0.000000],[0,0,-1,0],[9E+09,9E+09,9E+09,9E+09,9E+09,9E+09]];
    CONST robtarget T1610:=[[44.719878,72.512692,13.900025],[0.000000,0.000000,1.000000,0.000000],[0,0,-1,0],[9E+09,9E+09,9E+09,9E+09,9E+09,9E+09]];
    CONST robtarget T1611:=[[44.719878,44.587250,13.900025],[0.000000,0.000000,1.000000,0.000000],[0,0,-1,0],[9E+09,9E+09,9E+09,9E+09,9E+09,9E+09]];
    CONST robtarget T1612:=[[43.459873,45.884908,13.900025],[0.000000,0.000000,1.000000,0.000000],[0,0,-1,0],[9E+09,9E+09,9E+09,9E+09,9E+09,9E+09]];
    CONST robtarget T1613:=[[43.459873,72.670297,13.900025],[0.000000,0.000000,1.000000,0.000000],[0,0,-1,0],[9E+09,9E+09,9E+09,9E+09,9E+09,9E+09]];
    CONST robtarget T1614:=[[43.459873,87.329711,13.900025],[0.000000,0.000000,1.000000,0.000000],[0,0,-1,0],[9E+09,9E+09,9E+09,9E+09,9E+09,9E+09]];
    CONST robtarget T1615:=[[43.459873,114.115099,13.900025],[0.000000,0.000000,1.000000,0.000000],[0,0,-1,0],[9E+09,9E+09,9E+09,9E+09,9E+09,9E+09]];
    CONST robtarget T1616:=[[42.199869,112.721391,13.900025],[0.000000,0.000000,1.000000,0.000000],[0,0,-1,0],[9E+09,9E+09,9E+09,9E+09,9E+09,9E+09]];
    CONST robtarget T1617:=[[42.199869,86.948670,13.900025],[0.000000,0.000000,1.000000,0.000000],[0,0,-1,0],[9E+09,9E+09,9E+09,9E+09,9E+09,9E+09]];
    CONST robtarget T1618:=[[42.199869,73.051337,13.900025],[0.000000,0.000000,1.000000,0.000000],[0,0,-1,0],[9E+09,9E+09,9E+09,9E+09,9E+09,9E+09]];
    CONST robtarget T1619:=[[42.199869,47.278617,13.900025],[0.000000,0.000000,1.000000,0.000000],[0,0,-1,0],[9E+09,9E+09,9E+09,9E+09,9E+09,9E+09]];
    CONST robtarget T1620:=[[40.939864,48.787854,13.900025],[0.000000,0.000000,1.000000,0.000000],[0,0,-1,0],[9E+09,9E+09,9E+09,9E+09,9E+09,9E+09]];
    CONST robtarget T1621:=[[40.939864,73.708792,13.900025],[0.000000,0.000000,1.000000,0.000000],[0,0,-1,0],[9E+09,9E+09,9E+09,9E+09,9E+09,9E+09]];
    CONST robtarget T1622:=[[40.939864,86.291215,13.900025],[0.000000,0.000000,1.000000,0.000000],[0,0,-1,0],[9E+09,9E+09,9E+09,9E+09,9E+09,9E+09]];
    CONST robtarget T1623:=[[40.939864,111.212154,13.900025],[0.000000,0.000000,1.000000,0.000000],[0,0,-1,0],[9E+09,9E+09,9E+09,9E+09,9E+09,9E+09]];
    CONST robtarget T1624:=[[39.679860,109.560940,13.900025],[0.000000,0.000000,1.000000,0.000000],[0,0,-1,0],[9E+09,9E+09,9E+09,9E+09,9E+09,9E+09]];
    CONST robtarget T1625:=[[39.679860,85.271589,13.900025],[0.000000,0.000000,1.000000,0.000000],[0,0,-1,0],[9E+09,9E+09,9E+09,9E+09,9E+09,9E+09]];
    CONST robtarget T1626:=[[39.679860,74.728418,13.900025],[0.000000,0.000000,1.000000,0.000000],[0,0,-1,0],[9E+09,9E+09,9E+09,9E+09,9E+09,9E+09]];
    CONST robtarget T1627:=[[39.679860,50.439068,13.900025],[0.000000,0.000000,1.000000,0.000000],[0,0,-1,0],[9E+09,9E+09,9E+09,9E+09,9E+09,9E+09]];
    CONST robtarget T1628:=[[38.419855,52.240778,13.900025],[0.000000,0.000000,1.000000,0.000000],[0,0,-1,0],[9E+09,9E+09,9E+09,9E+09,9E+09,9E+09]];
    CONST robtarget T1629:=[[38.419855,76.422528,13.900025],[0.000000,0.000000,1.000000,0.000000],[0,0,-1,0],[9E+09,9E+09,9E+09,9E+09,9E+09,9E+09]];
    CONST robtarget T1630:=[[38.419855,83.577479,13.900025],[0.000000,0.000000,1.000000,0.000000],[0,0,-1,0],[9E+09,9E+09,9E+09,9E+09,9E+09,9E+09]];
    CONST robtarget T1631:=[[38.419855,107.759230,13.900025],[0.000000,0.000000,1.000000,0.000000],[0,0,-1,0],[9E+09,9E+09,9E+09,9E+09,9E+09,9E+09]];
    CONST robtarget T1632:=[[37.159851,105.775934,13.900025],[0.000000,0.000000,1.000000,0.000000],[0,0,-1,0],[9E+09,9E+09,9E+09,9E+09,9E+09,9E+09]];
    CONST robtarget T1633:=[[37.159851,54.224074,13.900025],[0.000000,0.000000,1.000000,0.000000],[0,0,-1,0],[9E+09,9E+09,9E+09,9E+09,9E+09,9E+09]];
    CONST robtarget T1634:=[[35.899846,56.444690,13.900025],[0.000000,0.000000,1.000000,0.000000],[0,0,-1,0],[9E+09,9E+09,9E+09,9E+09,9E+09,9E+09]];
    CONST robtarget T1635:=[[35.899846,103.555317,13.900025],[0.000000,0.000000,1.000000,0.000000],[0,0,-1,0],[9E+09,9E+09,9E+09,9E+09,9E+09,9E+09]];
    CONST robtarget T1636:=[[34.639842,101.007928,13.900025],[0.000000,0.000000,1.000000,0.000000],[0,0,-1,0],[9E+09,9E+09,9E+09,9E+09,9E+09,9E+09]];
    CONST robtarget T1637:=[[34.639842,58.992080,13.900025],[0.000000,0.000000,1.000000,0.000000],[0,0,-1,0],[9E+09,9E+09,9E+09,9E+09,9E+09,9E+09]];
    CONST robtarget T1638:=[[33.379837,61.953657,13.900025],[0.000000,0.000000,1.000000,0.000000],[0,0,-1,0],[9E+09,9E+09,9E+09,9E+09,9E+09,9E+09]];
    CONST robtarget T1639:=[[33.379837,98.046351,13.900025],[0.000000,0.000000,1.000000,0.000000],[0,0,-1,0],[9E+09,9E+09,9E+09,9E+09,9E+09,9E+09]];
    CONST robtarget T1640:=[[32.119833,94.360756,13.900025],[0.000000,0.000000,1.000000,0.000000],[0,0,-1,0],[9E+09,9E+09,9E+09,9E+09,9E+09,9E+09]];
    CONST robtarget T1641:=[[32.119833,65.639251,13.900025],[0.000000,0.000000,1.000000,0.000000],[0,0,-1,0],[9E+09,9E+09,9E+09,9E+09,9E+09,9E+09]];
    CONST robtarget T1642:=[[30.859828,70.797151,13.900025],[0.000000,0.000000,1.000000,0.000000],[0,0,-1,0],[9E+09,9E+09,9E+09,9E+09,9E+09,9E+09]];
    CONST robtarget T1643:=[[30.859828,89.202857,13.900025],[0.000000,0.000000,1.000000,0.000000],[0,0,-1,0],[9E+09,9E+09,9E+09,9E+09,9E+09,9E+09]];
    CONST robtarget T1644:=[[30.859828,70.797151,14.600035],[0.000000,0.000000,1.000000,0.000000],[0,0,-1,0],[9E+09,9E+09,9E+09,9E+09,9E+09,9E+09]];
    CONST robtarget T1645:=[[30.859828,89.202857,14.600035],[0.000000,0.000000,1.000000,0.000000],[0,0,-1,0],[9E+09,9E+09,9E+09,9E+09,9E+09,9E+09]];
    CONST robtarget T1646:=[[30.859828,70.797151,14.600035],[0.000000,0.000000,1.000000,0.000000],[0,0,-1,0],[9E+09,9E+09,9E+09,9E+09,9E+09,9E+09]];
    CONST robtarget T1647:=[[30.859828,89.202857,14.600035],[0.000000,0.000000,1.000000,0.000000],[0,0,-1,0],[9E+09,9E+09,9E+09,9E+09,9E+09,9E+09]];
    CONST robtarget T1648:=[[32.119833,94.360756,14.600035],[0.000000,0.000000,1.000000,0.000000],[0,0,-1,0],[9E+09,9E+09,9E+09,9E+09,9E+09,9E+09]];
    CONST robtarget T1649:=[[32.119833,65.639251,14.600035],[0.000000,0.000000,1.000000,0.000000],[0,0,-1,0],[9E+09,9E+09,9E+09,9E+09,9E+09,9E+09]];
    CONST robtarget T1650:=[[33.379837,61.953657,14.600035],[0.000000,0.000000,1.000000,0.000000],[0,0,-1,0],[9E+09,9E+09,9E+09,9E+09,9E+09,9E+09]];
    CONST robtarget T1651:=[[33.379837,98.046351,14.600035],[0.000000,0.000000,1.000000,0.000000],[0,0,-1,0],[9E+09,9E+09,9E+09,9E+09,9E+09,9E+09]];
    CONST robtarget T1652:=[[34.639842,101.007928,14.600035],[0.000000,0.000000,1.000000,0.000000],[0,0,-1,0],[9E+09,9E+09,9E+09,9E+09,9E+09,9E+09]];
    CONST robtarget T1653:=[[34.639842,58.992080,14.600035],[0.000000,0.000000,1.000000,0.000000],[0,0,-1,0],[9E+09,9E+09,9E+09,9E+09,9E+09,9E+09]];
    CONST robtarget T1654:=[[35.899846,56.444690,14.600035],[0.000000,0.000000,1.000000,0.000000],[0,0,-1,0],[9E+09,9E+09,9E+09,9E+09,9E+09,9E+09]];
    CONST robtarget T1655:=[[35.899846,103.555317,14.600035],[0.000000,0.000000,1.000000,0.000000],[0,0,-1,0],[9E+09,9E+09,9E+09,9E+09,9E+09,9E+09]];
    CONST robtarget T1656:=[[37.159851,105.775934,14.600035],[0.000000,0.000000,1.000000,0.000000],[0,0,-1,0],[9E+09,9E+09,9E+09,9E+09,9E+09,9E+09]];
    CONST robtarget T1657:=[[37.159851,54.224074,14.600035],[0.000000,0.000000,1.000000,0.000000],[0,0,-1,0],[9E+09,9E+09,9E+09,9E+09,9E+09,9E+09]];
    CONST robtarget T1658:=[[38.419855,52.240778,14.600035],[0.000000,0.000000,1.000000,0.000000],[0,0,-1,0],[9E+09,9E+09,9E+09,9E+09,9E+09,9E+09]];
    CONST robtarget T1659:=[[38.419855,76.422528,14.600035],[0.000000,0.000000,1.000000,0.000000],[0,0,-1,0],[9E+09,9E+09,9E+09,9E+09,9E+09,9E+09]];
    CONST robtarget T1660:=[[38.419855,83.577479,14.600035],[0.000000,0.000000,1.000000,0.000000],[0,0,-1,0],[9E+09,9E+09,9E+09,9E+09,9E+09,9E+09]];
    CONST robtarget T1661:=[[38.419855,107.759230,14.600035],[0.000000,0.000000,1.000000,0.000000],[0,0,-1,0],[9E+09,9E+09,9E+09,9E+09,9E+09,9E+09]];
    CONST robtarget T1662:=[[39.679860,109.560940,14.600035],[0.000000,0.000000,1.000000,0.000000],[0,0,-1,0],[9E+09,9E+09,9E+09,9E+09,9E+09,9E+09]];
    CONST robtarget T1663:=[[39.679860,85.271589,14.600035],[0.000000,0.000000,1.000000,0.000000],[0,0,-1,0],[9E+09,9E+09,9E+09,9E+09,9E+09,9E+09]];
    CONST robtarget T1664:=[[39.679860,74.728418,14.600035],[0.000000,0.000000,1.000000,0.000000],[0,0,-1,0],[9E+09,9E+09,9E+09,9E+09,9E+09,9E+09]];
    CONST robtarget T1665:=[[39.679860,50.439068,14.600035],[0.000000,0.000000,1.000000,0.000000],[0,0,-1,0],[9E+09,9E+09,9E+09,9E+09,9E+09,9E+09]];
    CONST robtarget T1666:=[[40.939864,48.787854,14.600035],[0.000000,0.000000,1.000000,0.000000],[0,0,-1,0],[9E+09,9E+09,9E+09,9E+09,9E+09,9E+09]];
    CONST robtarget T1667:=[[40.939864,73.708792,14.600035],[0.000000,0.000000,1.000000,0.000000],[0,0,-1,0],[9E+09,9E+09,9E+09,9E+09,9E+09,9E+09]];
    CONST robtarget T1668:=[[40.939864,86.291215,14.600035],[0.000000,0.000000,1.000000,0.000000],[0,0,-1,0],[9E+09,9E+09,9E+09,9E+09,9E+09,9E+09]];
    CONST robtarget T1669:=[[40.939864,111.212154,14.600035],[0.000000,0.000000,1.000000,0.000000],[0,0,-1,0],[9E+09,9E+09,9E+09,9E+09,9E+09,9E+09]];
    CONST robtarget T1670:=[[42.199869,112.721391,14.600035],[0.000000,0.000000,1.000000,0.000000],[0,0,-1,0],[9E+09,9E+09,9E+09,9E+09,9E+09,9E+09]];
    CONST robtarget T1671:=[[42.199869,86.948670,14.600035],[0.000000,0.000000,1.000000,0.000000],[0,0,-1,0],[9E+09,9E+09,9E+09,9E+09,9E+09,9E+09]];
    CONST robtarget T1672:=[[42.199869,73.051337,14.600035],[0.000000,0.000000,1.000000,0.000000],[0,0,-1,0],[9E+09,9E+09,9E+09,9E+09,9E+09,9E+09]];
    CONST robtarget T1673:=[[42.199869,47.278617,14.600035],[0.000000,0.000000,1.000000,0.000000],[0,0,-1,0],[9E+09,9E+09,9E+09,9E+09,9E+09,9E+09]];
    CONST robtarget T1674:=[[43.459873,45.884908,14.600035],[0.000000,0.000000,1.000000,0.000000],[0,0,-1,0],[9E+09,9E+09,9E+09,9E+09,9E+09,9E+09]];
    CONST robtarget T1675:=[[43.459873,72.670297,14.600035],[0.000000,0.000000,1.000000,0.000000],[0,0,-1,0],[9E+09,9E+09,9E+09,9E+09,9E+09,9E+09]];
    CONST robtarget T1676:=[[43.459873,87.329711,14.600035],[0.000000,0.000000,1.000000,0.000000],[0,0,-1,0],[9E+09,9E+09,9E+09,9E+09,9E+09,9E+09]];
    CONST robtarget T1677:=[[43.459873,114.115099,14.600035],[0.000000,0.000000,1.000000,0.000000],[0,0,-1,0],[9E+09,9E+09,9E+09,9E+09,9E+09,9E+09]];
    CONST robtarget T1678:=[[44.719878,115.412758,14.600035],[0.000000,0.000000,1.000000,0.000000],[0,0,-1,0],[9E+09,9E+09,9E+09,9E+09,9E+09,9E+09]];
    CONST robtarget T1679:=[[44.719878,87.487316,14.600035],[0.000000,0.000000,1.000000,0.000000],[0,0,-1,0],[9E+09,9E+09,9E+09,9E+09,9E+09,9E+09]];
    CONST robtarget T1680:=[[44.719878,72.512692,14.600035],[0.000000,0.000000,1.000000,0.000000],[0,0,-1,0],[9E+09,9E+09,9E+09,9E+09,9E+09,9E+09]];
    CONST robtarget T1681:=[[44.719878,44.587250,14.600035],[0.000000,0.000000,1.000000,0.000000],[0,0,-1,0],[9E+09,9E+09,9E+09,9E+09,9E+09,9E+09]];
    CONST robtarget T1682:=[[45.979882,43.373063,14.600035],[0.000000,0.000000,1.000000,0.000000],[0,0,-1,0],[9E+09,9E+09,9E+09,9E+09,9E+09,9E+09]];
    CONST robtarget T1683:=[[45.979882,72.576253,14.600035],[0.000000,0.000000,1.000000,0.000000],[0,0,-1,0],[9E+09,9E+09,9E+09,9E+09,9E+09,9E+09]];
    CONST robtarget T1684:=[[45.979882,87.423755,14.600035],[0.000000,0.000000,1.000000,0.000000],[0,0,-1,0],[9E+09,9E+09,9E+09,9E+09,9E+09,9E+09]];
    CONST robtarget T1685:=[[45.979882,116.626944,14.600035],[0.000000,0.000000,1.000000,0.000000],[0,0,-1,0],[9E+09,9E+09,9E+09,9E+09,9E+09,9E+09]];
    CONST robtarget T1686:=[[47.239887,117.767805,14.600035],[0.000000,0.000000,1.000000,0.000000],[0,0,-1,0],[9E+09,9E+09,9E+09,9E+09,9E+09,9E+09]];
    CONST robtarget T1687:=[[47.239887,87.152583,14.600035],[0.000000,0.000000,1.000000,0.000000],[0,0,-1,0],[9E+09,9E+09,9E+09,9E+09,9E+09,9E+09]];
    CONST robtarget T1688:=[[47.239887,72.847425,14.600035],[0.000000,0.000000,1.000000,0.000000],[0,0,-1,0],[9E+09,9E+09,9E+09,9E+09,9E+09,9E+09]];
    CONST robtarget T1689:=[[47.239887,42.232203,14.600035],[0.000000,0.000000,1.000000,0.000000],[0,0,-1,0],[9E+09,9E+09,9E+09,9E+09,9E+09,9E+09]];
    CONST robtarget T1690:=[[48.499891,41.180273,14.600035],[0.000000,0.000000,1.000000,0.000000],[0,0,-1,0],[9E+09,9E+09,9E+09,9E+09,9E+09,9E+09]];
    CONST robtarget T1691:=[[48.499891,73.379202,14.600035],[0.000000,0.000000,1.000000,0.000000],[0,0,-1,0],[9E+09,9E+09,9E+09,9E+09,9E+09,9E+09]];
    CONST robtarget T1692:=[[48.499891,86.620805,14.600035],[0.000000,0.000000,1.000000,0.000000],[0,0,-1,0],[9E+09,9E+09,9E+09,9E+09,9E+09,9E+09]];
    CONST robtarget T1693:=[[48.499891,118.819735,14.600035],[0.000000,0.000000,1.000000,0.000000],[0,0,-1,0],[9E+09,9E+09,9E+09,9E+09,9E+09,9E+09]];
    CONST robtarget T1694:=[[49.759896,119.803025,14.600035],[0.000000,0.000000,1.000000,0.000000],[0,0,-1,0],[9E+09,9E+09,9E+09,9E+09,9E+09,9E+09]];
    CONST robtarget T1695:=[[49.759896,85.779969,14.600035],[0.000000,0.000000,1.000000,0.000000],[0,0,-1,0],[9E+09,9E+09,9E+09,9E+09,9E+09,9E+09]];
    CONST robtarget T1696:=[[49.759896,74.220038,14.600035],[0.000000,0.000000,1.000000,0.000000],[0,0,-1,0],[9E+09,9E+09,9E+09,9E+09,9E+09,9E+09]];
    CONST robtarget T1697:=[[49.759896,40.196983,14.600035],[0.000000,0.000000,1.000000,0.000000],[0,0,-1,0],[9E+09,9E+09,9E+09,9E+09,9E+09,9E+09]];
    CONST robtarget T1698:=[[51.019900,39.265681,14.600035],[0.000000,0.000000,1.000000,0.000000],[0,0,-1,0],[9E+09,9E+09,9E+09,9E+09,9E+09,9E+09]];
    CONST robtarget T1699:=[[51.019900,75.547902,14.600035],[0.000000,0.000000,1.000000,0.000000],[0,0,-1,0],[9E+09,9E+09,9E+09,9E+09,9E+09,9E+09]];
    CONST robtarget T1700:=[[51.019900,84.452106,14.600035],[0.000000,0.000000,1.000000,0.000000],[0,0,-1,0],[9E+09,9E+09,9E+09,9E+09,9E+09,9E+09]];
    CONST robtarget T1701:=[[51.019900,120.734326,14.600035],[0.000000,0.000000,1.000000,0.000000],[0,0,-1,0],[9E+09,9E+09,9E+09,9E+09,9E+09,9E+09]];
    CONST robtarget T1702:=[[52.279905,121.607260,14.600035],[0.000000,0.000000,1.000000,0.000000],[0,0,-1,0],[9E+09,9E+09,9E+09,9E+09,9E+09,9E+09]];
    CONST robtarget T1703:=[[52.279905,81.789524,14.600035],[0.000000,0.000000,1.000000,0.000000],[0,0,-1,0],[9E+09,9E+09,9E+09,9E+09,9E+09,9E+09]];
    CONST robtarget T1704:=[[52.279905,78.210483,14.600035],[0.000000,0.000000,1.000000,0.000000],[0,0,-1,0],[9E+09,9E+09,9E+09,9E+09,9E+09,9E+09]];
    CONST robtarget T1705:=[[52.279905,38.392748,14.600035],[0.000000,0.000000,1.000000,0.000000],[0,0,-1,0],[9E+09,9E+09,9E+09,9E+09,9E+09,9E+09]];
    CONST robtarget T1706:=[[53.539909,37.589739,14.600035],[0.000000,0.000000,1.000000,0.000000],[0,0,-1,0],[9E+09,9E+09,9E+09,9E+09,9E+09,9E+09]];
    CONST robtarget T1707:=[[53.539909,122.410268,14.600035],[0.000000,0.000000,1.000000,0.000000],[0,0,-1,0],[9E+09,9E+09,9E+09,9E+09,9E+09,9E+09]];
    CONST robtarget T1708:=[[54.799914,123.174878,14.600035],[0.000000,0.000000,1.000000,0.000000],[0,0,-1,0],[9E+09,9E+09,9E+09,9E+09,9E+09,9E+09]];
    CONST robtarget T1709:=[[54.799914,36.825129,14.600035],[0.000000,0.000000,1.000000,0.000000],[0,0,-1,0],[9E+09,9E+09,9E+09,9E+09,9E+09,9E+09]];
    CONST robtarget T1710:=[[56.059918,36.110177,14.600035],[0.000000,0.000000,1.000000,0.000000],[0,0,-1,0],[9E+09,9E+09,9E+09,9E+09,9E+09,9E+09]];
    CONST robtarget T1711:=[[56.059918,123.889831,14.600035],[0.000000,0.000000,1.000000,0.000000],[0,0,-1,0],[9E+09,9E+09,9E+09,9E+09,9E+09,9E+09]];
    CONST robtarget T1712:=[[57.319923,124.546114,14.600035],[0.000000,0.000000,1.000000,0.000000],[0,0,-1,0],[9E+09,9E+09,9E+09,9E+09,9E+09,9E+09]];
    CONST robtarget T1713:=[[57.319923,35.453894,14.600035],[0.000000,0.000000,1.000000,0.000000],[0,0,-1,0],[9E+09,9E+09,9E+09,9E+09,9E+09,9E+09]];
    CONST robtarget T1714:=[[58.579927,34.827050,14.600035],[0.000000,0.000000,1.000000,0.000000],[0,0,-1,0],[9E+09,9E+09,9E+09,9E+09,9E+09,9E+09]];
    CONST robtarget T1715:=[[58.579927,125.172958,14.600035],[0.000000,0.000000,1.000000,0.000000],[0,0,-1,0],[9E+09,9E+09,9E+09,9E+09,9E+09,9E+09]];
    CONST robtarget T1716:=[[59.839932,125.745278,14.600035],[0.000000,0.000000,1.000000,0.000000],[0,0,-1,0],[9E+09,9E+09,9E+09,9E+09,9E+09,9E+09]];
    CONST robtarget T1717:=[[59.839932,34.254730,14.600035],[0.000000,0.000000,1.000000,0.000000],[0,0,-1,0],[9E+09,9E+09,9E+09,9E+09,9E+09,9E+09]];
    CONST robtarget T1718:=[[61.099936,33.722290,14.600035],[0.000000,0.000000,1.000000,0.000000],[0,0,-1,0],[9E+09,9E+09,9E+09,9E+09,9E+09,9E+09]];
    CONST robtarget T1719:=[[61.099936,126.277717,14.600035],[0.000000,0.000000,1.000000,0.000000],[0,0,-1,0],[9E+09,9E+09,9E+09,9E+09,9E+09,9E+09]];
    CONST robtarget T1720:=[[62.359941,126.783143,14.600035],[0.000000,0.000000,1.000000,0.000000],[0,0,-1,0],[9E+09,9E+09,9E+09,9E+09,9E+09,9E+09]];
    CONST robtarget T1721:=[[62.359941,33.216864,14.600035],[0.000000,0.000000,1.000000,0.000000],[0,0,-1,0],[9E+09,9E+09,9E+09,9E+09,9E+09,9E+09]];
    CONST robtarget T1722:=[[63.619945,32.772318,14.600035],[0.000000,0.000000,1.000000,0.000000],[0,0,-1,0],[9E+09,9E+09,9E+09,9E+09,9E+09,9E+09]];
    CONST robtarget T1723:=[[63.619945,127.227690,14.600035],[0.000000,0.000000,1.000000,0.000000],[0,0,-1,0],[9E+09,9E+09,9E+09,9E+09,9E+09,9E+09]];
    CONST robtarget T1724:=[[64.879950,127.652167,14.600035],[0.000000,0.000000,1.000000,0.000000],[0,0,-1,0],[9E+09,9E+09,9E+09,9E+09,9E+09,9E+09]];
    CONST robtarget T1725:=[[64.879950,32.347841,14.600035],[0.000000,0.000000,1.000000,0.000000],[0,0,-1,0],[9E+09,9E+09,9E+09,9E+09,9E+09,9E+09]];
    CONST robtarget T1726:=[[66.139954,31.969479,14.600035],[0.000000,0.000000,1.000000,0.000000],[0,0,-1,0],[9E+09,9E+09,9E+09,9E+09,9E+09,9E+09]];
    CONST robtarget T1727:=[[66.139954,128.030529,14.600035],[0.000000,0.000000,1.000000,0.000000],[0,0,-1,0],[9E+09,9E+09,9E+09,9E+09,9E+09,9E+09]];
    CONST robtarget T1728:=[[67.399959,128.374988,14.600035],[0.000000,0.000000,1.000000,0.000000],[0,0,-1,0],[9E+09,9E+09,9E+09,9E+09,9E+09,9E+09]];
    CONST robtarget T1729:=[[67.399959,31.625019,14.600035],[0.000000,0.000000,1.000000,0.000000],[0,0,-1,0],[9E+09,9E+09,9E+09,9E+09,9E+09,9E+09]];
    CONST robtarget T1730:=[[68.659963,31.307526,14.600035],[0.000000,0.000000,1.000000,0.000000],[0,0,-1,0],[9E+09,9E+09,9E+09,9E+09,9E+09,9E+09]];
    CONST robtarget T1731:=[[68.659963,128.692481,14.600035],[0.000000,0.000000,1.000000,0.000000],[0,0,-1,0],[9E+09,9E+09,9E+09,9E+09,9E+09,9E+09]];
    CONST robtarget T1732:=[[69.919968,128.960575,14.600035],[0.000000,0.000000,1.000000,0.000000],[0,0,-1,0],[9E+09,9E+09,9E+09,9E+09,9E+09,9E+09]];
    CONST robtarget T1733:=[[69.919968,31.039433,14.600035],[0.000000,0.000000,1.000000,0.000000],[0,0,-1,0],[9E+09,9E+09,9E+09,9E+09,9E+09,9E+09]];
    CONST robtarget T1734:=[[71.179972,30.786444,14.600035],[0.000000,0.000000,1.000000,0.000000],[0,0,-1,0],[9E+09,9E+09,9E+09,9E+09,9E+09,9E+09]];
    CONST robtarget T1735:=[[71.179972,129.213563,14.600035],[0.000000,0.000000,1.000000,0.000000],[0,0,-1,0],[9E+09,9E+09,9E+09,9E+09,9E+09,9E+09]];
    CONST robtarget T1736:=[[72.439977,129.413129,14.600035],[0.000000,0.000000,1.000000,0.000000],[0,0,-1,0],[9E+09,9E+09,9E+09,9E+09,9E+09,9E+09]];
    CONST robtarget T1737:=[[72.439977,83.409593,14.600035],[0.000000,0.000000,1.000000,0.000000],[0,0,-1,0],[9E+09,9E+09,9E+09,9E+09,9E+09,9E+09]];
    CONST robtarget T1738:=[[72.439977,76.590415,14.600035],[0.000000,0.000000,1.000000,0.000000],[0,0,-1,0],[9E+09,9E+09,9E+09,9E+09,9E+09,9E+09]];
    CONST robtarget T1739:=[[72.439977,30.586879,14.600035],[0.000000,0.000000,1.000000,0.000000],[0,0,-1,0],[9E+09,9E+09,9E+09,9E+09,9E+09,9E+09]];
    CONST robtarget T1740:=[[73.699981,30.406130,14.600035],[0.000000,0.000000,1.000000,0.000000],[0,0,-1,0],[9E+09,9E+09,9E+09,9E+09,9E+09,9E+09]];
    CONST robtarget T1741:=[[73.699981,40.937335,14.600035],[0.000000,0.000000,1.000000,0.000000],[0,0,-1,0],[9E+09,9E+09,9E+09,9E+09,9E+09,9E+09]];
    CONST robtarget T1742:=[[73.699981,49.062665,14.600035],[0.000000,0.000000,1.000000,0.000000],[0,0,-1,0],[9E+09,9E+09,9E+09,9E+09,9E+09,9E+09]];
    CONST robtarget T1743:=[[73.699981,74.600294,14.600035],[0.000000,0.000000,1.000000,0.000000],[0,0,-1,0],[9E+09,9E+09,9E+09,9E+09,9E+09,9E+09]];
    CONST robtarget T1744:=[[73.699981,85.399713,14.600035],[0.000000,0.000000,1.000000,0.000000],[0,0,-1,0],[9E+09,9E+09,9E+09,9E+09,9E+09,9E+09]];
    CONST robtarget T1745:=[[73.699981,110.937342,14.600035],[0.000000,0.000000,1.000000,0.000000],[0,0,-1,0],[9E+09,9E+09,9E+09,9E+09,9E+09,9E+09]];
    CONST robtarget T1746:=[[73.699981,119.062672,14.600035],[0.000000,0.000000,1.000000,0.000000],[0,0,-1,0],[9E+09,9E+09,9E+09,9E+09,9E+09,9E+09]];
    CONST robtarget T1747:=[[73.699981,129.593877,14.600035],[0.000000,0.000000,1.000000,0.000000],[0,0,-1,0],[9E+09,9E+09,9E+09,9E+09,9E+09,9E+09]];
    CONST robtarget T1748:=[[74.959986,129.735844,14.600035],[0.000000,0.000000,1.000000,0.000000],[0,0,-1,0],[9E+09,9E+09,9E+09,9E+09,9E+09,9E+09]];
    CONST robtarget T1749:=[[74.959986,120.544921,14.600035],[0.000000,0.000000,1.000000,0.000000],[0,0,-1,0],[9E+09,9E+09,9E+09,9E+09,9E+09,9E+09]];
    CONST robtarget T1750:=[[74.959986,109.455091,14.600035],[0.000000,0.000000,1.000000,0.000000],[0,0,-1,0],[9E+09,9E+09,9E+09,9E+09,9E+09,9E+09]];
    CONST robtarget T1751:=[[74.959986,86.587380,14.600035],[0.000000,0.000000,1.000000,0.000000],[0,0,-1,0],[9E+09,9E+09,9E+09,9E+09,9E+09,9E+09]];
    CONST robtarget T1752:=[[74.959986,73.412627,14.600035],[0.000000,0.000000,1.000000,0.000000],[0,0,-1,0],[9E+09,9E+09,9E+09,9E+09,9E+09,9E+09]];
    CONST robtarget T1753:=[[74.959986,50.544916,14.600035],[0.000000,0.000000,1.000000,0.000000],[0,0,-1,0],[9E+09,9E+09,9E+09,9E+09,9E+09,9E+09]];
    CONST robtarget T1754:=[[74.959986,39.455086,14.600035],[0.000000,0.000000,1.000000,0.000000],[0,0,-1,0],[9E+09,9E+09,9E+09,9E+09,9E+09,9E+09]];
    CONST robtarget T1755:=[[74.959986,30.264163,14.600035],[0.000000,0.000000,1.000000,0.000000],[0,0,-1,0],[9E+09,9E+09,9E+09,9E+09,9E+09,9E+09]];
    CONST robtarget T1756:=[[76.219990,30.153959,14.600035],[0.000000,0.000000,1.000000,0.000000],[0,0,-1,0],[9E+09,9E+09,9E+09,9E+09,9E+09,9E+09]];
    CONST robtarget T1757:=[[76.219990,38.524551,14.600035],[0.000000,0.000000,1.000000,0.000000],[0,0,-1,0],[9E+09,9E+09,9E+09,9E+09,9E+09,9E+09]];
    CONST robtarget T1758:=[[76.219990,51.475451,14.600035],[0.000000,0.000000,1.000000,0.000000],[0,0,-1,0],[9E+09,9E+09,9E+09,9E+09,9E+09,9E+09]];
    CONST robtarget T1759:=[[76.219990,72.623502,14.600035],[0.000000,0.000000,1.000000,0.000000],[0,0,-1,0],[9E+09,9E+09,9E+09,9E+09,9E+09,9E+09]];
    CONST robtarget T1760:=[[76.219990,87.376506,14.600035],[0.000000,0.000000,1.000000,0.000000],[0,0,-1,0],[9E+09,9E+09,9E+09,9E+09,9E+09,9E+09]];
    CONST robtarget T1761:=[[76.219990,108.524556,14.600035],[0.000000,0.000000,1.000000,0.000000],[0,0,-1,0],[9E+09,9E+09,9E+09,9E+09,9E+09,9E+09]];
    CONST robtarget T1762:=[[76.219990,121.475457,14.600035],[0.000000,0.000000,1.000000,0.000000],[0,0,-1,0],[9E+09,9E+09,9E+09,9E+09,9E+09,9E+09]];
    CONST robtarget T1763:=[[76.219990,129.846049,14.600035],[0.000000,0.000000,1.000000,0.000000],[0,0,-1,0],[9E+09,9E+09,9E+09,9E+09,9E+09,9E+09]];
    CONST robtarget T1764:=[[77.479995,129.931001,14.600035],[0.000000,0.000000,1.000000,0.000000],[0,0,-1,0],[9E+09,9E+09,9E+09,9E+09,9E+09,9E+09]];
    CONST robtarget T1765:=[[77.479995,122.050628,14.600035],[0.000000,0.000000,1.000000,0.000000],[0,0,-1,0],[9E+09,9E+09,9E+09,9E+09,9E+09,9E+09]];
    CONST robtarget T1766:=[[77.479995,107.949384,14.600035],[0.000000,0.000000,1.000000,0.000000],[0,0,-1,0],[9E+09,9E+09,9E+09,9E+09,9E+09,9E+09]];
    CONST robtarget T1767:=[[77.479995,87.904989,14.600035],[0.000000,0.000000,1.000000,0.000000],[0,0,-1,0],[9E+09,9E+09,9E+09,9E+09,9E+09,9E+09]];
    CONST robtarget T1768:=[[77.479995,72.095019,14.600035],[0.000000,0.000000,1.000000,0.000000],[0,0,-1,0],[9E+09,9E+09,9E+09,9E+09,9E+09,9E+09]];
    CONST robtarget T1769:=[[77.479995,52.050624,14.600035],[0.000000,0.000000,1.000000,0.000000],[0,0,-1,0],[9E+09,9E+09,9E+09,9E+09,9E+09,9E+09]];
    CONST robtarget T1770:=[[77.479995,37.949379,14.600035],[0.000000,0.000000,1.000000,0.000000],[0,0,-1,0],[9E+09,9E+09,9E+09,9E+09,9E+09,9E+09]];
    CONST robtarget T1771:=[[77.479995,30.069007,14.600035],[0.000000,0.000000,1.000000,0.000000],[0,0,-1,0],[9E+09,9E+09,9E+09,9E+09,9E+09,9E+09]];
    CONST robtarget T1772:=[[78.739999,30.028279,14.600035],[0.000000,0.000000,1.000000,0.000000],[0,0,-1,0],[9E+09,9E+09,9E+09,9E+09,9E+09,9E+09]];
    CONST robtarget T1773:=[[78.739999,37.608991,14.600035],[0.000000,0.000000,1.000000,0.000000],[0,0,-1,0],[9E+09,9E+09,9E+09,9E+09,9E+09,9E+09]];
    CONST robtarget T1774:=[[78.739999,52.391011,14.600035],[0.000000,0.000000,1.000000,0.000000],[0,0,-1,0],[9E+09,9E+09,9E+09,9E+09,9E+09,9E+09]];
    CONST robtarget T1775:=[[78.739999,71.801996,14.600035],[0.000000,0.000000,1.000000,0.000000],[0,0,-1,0],[9E+09,9E+09,9E+09,9E+09,9E+09,9E+09]];
    CONST robtarget T1776:=[[78.739999,88.198011,14.600035],[0.000000,0.000000,1.000000,0.000000],[0,0,-1,0],[9E+09,9E+09,9E+09,9E+09,9E+09,9E+09]];
    CONST robtarget T1777:=[[78.739999,107.608996,14.600035],[0.000000,0.000000,1.000000,0.000000],[0,0,-1,0],[9E+09,9E+09,9E+09,9E+09,9E+09,9E+09]];
    CONST robtarget T1778:=[[78.739999,122.391017,14.600035],[0.000000,0.000000,1.000000,0.000000],[0,0,-1,0],[9E+09,9E+09,9E+09,9E+09,9E+09,9E+09]];
    CONST robtarget T1779:=[[78.739999,129.971729,14.600035],[0.000000,0.000000,1.000000,0.000000],[0,0,-1,0],[9E+09,9E+09,9E+09,9E+09,9E+09,9E+09]];
    CONST robtarget T1780:=[[80.000004,130.000008,14.600035],[0.000000,0.000000,1.000000,0.000000],[0,0,-1,0],[9E+09,9E+09,9E+09,9E+09,9E+09,9E+09]];
    CONST robtarget T1781:=[[80.000004,122.487319,14.600035],[0.000000,0.000000,1.000000,0.000000],[0,0,-1,0],[9E+09,9E+09,9E+09,9E+09,9E+09,9E+09]];
    CONST robtarget T1782:=[[80.000004,107.512696,14.600035],[0.000000,0.000000,1.000000,0.000000],[0,0,-1,0],[9E+09,9E+09,9E+09,9E+09,9E+09,9E+09]];
    CONST robtarget T1783:=[[80.000004,88.292469,14.600035],[0.000000,0.000000,1.000000,0.000000],[0,0,-1,0],[9E+09,9E+09,9E+09,9E+09,9E+09,9E+09]];
    CONST robtarget T1784:=[[80.000004,71.707538,14.600035],[0.000000,0.000000,1.000000,0.000000],[0,0,-1,0],[9E+09,9E+09,9E+09,9E+09,9E+09,9E+09]];
    CONST robtarget T1785:=[[80.000004,52.487312,14.600035],[0.000000,0.000000,1.000000,0.000000],[0,0,-1,0],[9E+09,9E+09,9E+09,9E+09,9E+09,9E+09]];
    CONST robtarget T1786:=[[80.000004,37.512688,14.600035],[0.000000,0.000000,1.000000,0.000000],[0,0,-1,0],[9E+09,9E+09,9E+09,9E+09,9E+09,9E+09]];
    CONST robtarget T1787:=[[80.000004,30.000000,14.600035],[0.000000,0.000000,1.000000,0.000000],[0,0,-1,0],[9E+09,9E+09,9E+09,9E+09,9E+09,9E+09]];
    CONST robtarget T1788:=[[81.260008,30.028279,14.600035],[0.000000,0.000000,1.000000,0.000000],[0,0,-1,0],[9E+09,9E+09,9E+09,9E+09,9E+09,9E+09]];
    CONST robtarget T1789:=[[81.260008,37.608991,14.600035],[0.000000,0.000000,1.000000,0.000000],[0,0,-1,0],[9E+09,9E+09,9E+09,9E+09,9E+09,9E+09]];
    CONST robtarget T1790:=[[81.260008,52.391011,14.600035],[0.000000,0.000000,1.000000,0.000000],[0,0,-1,0],[9E+09,9E+09,9E+09,9E+09,9E+09,9E+09]];
    CONST robtarget T1791:=[[81.260008,71.801996,14.600035],[0.000000,0.000000,1.000000,0.000000],[0,0,-1,0],[9E+09,9E+09,9E+09,9E+09,9E+09,9E+09]];
    CONST robtarget T1792:=[[81.260008,88.198011,14.600035],[0.000000,0.000000,1.000000,0.000000],[0,0,-1,0],[9E+09,9E+09,9E+09,9E+09,9E+09,9E+09]];
    CONST robtarget T1793:=[[81.260008,107.608996,14.600035],[0.000000,0.000000,1.000000,0.000000],[0,0,-1,0],[9E+09,9E+09,9E+09,9E+09,9E+09,9E+09]];
    CONST robtarget T1794:=[[81.260008,122.391017,14.600035],[0.000000,0.000000,1.000000,0.000000],[0,0,-1,0],[9E+09,9E+09,9E+09,9E+09,9E+09,9E+09]];
    CONST robtarget T1795:=[[81.260008,129.971729,14.600035],[0.000000,0.000000,1.000000,0.000000],[0,0,-1,0],[9E+09,9E+09,9E+09,9E+09,9E+09,9E+09]];
    CONST robtarget T1796:=[[82.520013,129.931001,14.600035],[0.000000,0.000000,1.000000,0.000000],[0,0,-1,0],[9E+09,9E+09,9E+09,9E+09,9E+09,9E+09]];
    CONST robtarget T1797:=[[82.520013,122.050628,14.600035],[0.000000,0.000000,1.000000,0.000000],[0,0,-1,0],[9E+09,9E+09,9E+09,9E+09,9E+09,9E+09]];
    CONST robtarget T1798:=[[82.520013,107.949384,14.600035],[0.000000,0.000000,1.000000,0.000000],[0,0,-1,0],[9E+09,9E+09,9E+09,9E+09,9E+09,9E+09]];
    CONST robtarget T1799:=[[82.520013,87.904989,14.600035],[0.000000,0.000000,1.000000,0.000000],[0,0,-1,0],[9E+09,9E+09,9E+09,9E+09,9E+09,9E+09]];
    CONST robtarget T1800:=[[82.520013,72.095019,14.600035],[0.000000,0.000000,1.000000,0.000000],[0,0,-1,0],[9E+09,9E+09,9E+09,9E+09,9E+09,9E+09]];
    CONST robtarget T1801:=[[82.520013,52.050624,14.600035],[0.000000,0.000000,1.000000,0.000000],[0,0,-1,0],[9E+09,9E+09,9E+09,9E+09,9E+09,9E+09]];
    CONST robtarget T1802:=[[82.520013,37.949379,14.600035],[0.000000,0.000000,1.000000,0.000000],[0,0,-1,0],[9E+09,9E+09,9E+09,9E+09,9E+09,9E+09]];
    CONST robtarget T1803:=[[82.520013,30.069007,14.600035],[0.000000,0.000000,1.000000,0.000000],[0,0,-1,0],[9E+09,9E+09,9E+09,9E+09,9E+09,9E+09]];
    CONST robtarget T1804:=[[83.780017,30.153959,14.600035],[0.000000,0.000000,1.000000,0.000000],[0,0,-1,0],[9E+09,9E+09,9E+09,9E+09,9E+09,9E+09]];
    CONST robtarget T1805:=[[83.780017,38.524551,14.600035],[0.000000,0.000000,1.000000,0.000000],[0,0,-1,0],[9E+09,9E+09,9E+09,9E+09,9E+09,9E+09]];
    CONST robtarget T1806:=[[83.780017,51.475451,14.600035],[0.000000,0.000000,1.000000,0.000000],[0,0,-1,0],[9E+09,9E+09,9E+09,9E+09,9E+09,9E+09]];
    CONST robtarget T1807:=[[83.780017,72.623502,14.600035],[0.000000,0.000000,1.000000,0.000000],[0,0,-1,0],[9E+09,9E+09,9E+09,9E+09,9E+09,9E+09]];
    CONST robtarget T1808:=[[83.780017,87.376506,14.600035],[0.000000,0.000000,1.000000,0.000000],[0,0,-1,0],[9E+09,9E+09,9E+09,9E+09,9E+09,9E+09]];
    CONST robtarget T1809:=[[83.780017,108.524556,14.600035],[0.000000,0.000000,1.000000,0.000000],[0,0,-1,0],[9E+09,9E+09,9E+09,9E+09,9E+09,9E+09]];
    CONST robtarget T1810:=[[83.780017,121.475457,14.600035],[0.000000,0.000000,1.000000,0.000000],[0,0,-1,0],[9E+09,9E+09,9E+09,9E+09,9E+09,9E+09]];
    CONST robtarget T1811:=[[83.780017,129.846049,14.600035],[0.000000,0.000000,1.000000,0.000000],[0,0,-1,0],[9E+09,9E+09,9E+09,9E+09,9E+09,9E+09]];
    CONST robtarget T1812:=[[85.040022,129.735844,14.600035],[0.000000,0.000000,1.000000,0.000000],[0,0,-1,0],[9E+09,9E+09,9E+09,9E+09,9E+09,9E+09]];
    CONST robtarget T1813:=[[85.040022,120.544921,14.600035],[0.000000,0.000000,1.000000,0.000000],[0,0,-1,0],[9E+09,9E+09,9E+09,9E+09,9E+09,9E+09]];
    CONST robtarget T1814:=[[85.040022,109.455091,14.600035],[0.000000,0.000000,1.000000,0.000000],[0,0,-1,0],[9E+09,9E+09,9E+09,9E+09,9E+09,9E+09]];
    CONST robtarget T1815:=[[85.040022,86.587380,14.600035],[0.000000,0.000000,1.000000,0.000000],[0,0,-1,0],[9E+09,9E+09,9E+09,9E+09,9E+09,9E+09]];
    CONST robtarget T1816:=[[85.040022,73.412627,14.600035],[0.000000,0.000000,1.000000,0.000000],[0,0,-1,0],[9E+09,9E+09,9E+09,9E+09,9E+09,9E+09]];
    CONST robtarget T1817:=[[85.040022,50.544916,14.600035],[0.000000,0.000000,1.000000,0.000000],[0,0,-1,0],[9E+09,9E+09,9E+09,9E+09,9E+09,9E+09]];
    CONST robtarget T1818:=[[85.040022,39.455086,14.600035],[0.000000,0.000000,1.000000,0.000000],[0,0,-1,0],[9E+09,9E+09,9E+09,9E+09,9E+09,9E+09]];
    CONST robtarget T1819:=[[85.040022,30.264163,14.600035],[0.000000,0.000000,1.000000,0.000000],[0,0,-1,0],[9E+09,9E+09,9E+09,9E+09,9E+09,9E+09]];
    CONST robtarget T1820:=[[86.300026,30.406130,14.600035],[0.000000,0.000000,1.000000,0.000000],[0,0,-1,0],[9E+09,9E+09,9E+09,9E+09,9E+09,9E+09]];
    CONST robtarget T1821:=[[86.300026,40.937335,14.600035],[0.000000,0.000000,1.000000,0.000000],[0,0,-1,0],[9E+09,9E+09,9E+09,9E+09,9E+09,9E+09]];
    CONST robtarget T1822:=[[86.300026,49.062665,14.600035],[0.000000,0.000000,1.000000,0.000000],[0,0,-1,0],[9E+09,9E+09,9E+09,9E+09,9E+09,9E+09]];
    CONST robtarget T1823:=[[86.300026,74.600294,14.600035],[0.000000,0.000000,1.000000,0.000000],[0,0,-1,0],[9E+09,9E+09,9E+09,9E+09,9E+09,9E+09]];
    CONST robtarget T1824:=[[86.300026,85.399713,14.600035],[0.000000,0.000000,1.000000,0.000000],[0,0,-1,0],[9E+09,9E+09,9E+09,9E+09,9E+09,9E+09]];
    CONST robtarget T1825:=[[86.300026,110.937342,14.600035],[0.000000,0.000000,1.000000,0.000000],[0,0,-1,0],[9E+09,9E+09,9E+09,9E+09,9E+09,9E+09]];
    CONST robtarget T1826:=[[86.300026,119.062672,14.600035],[0.000000,0.000000,1.000000,0.000000],[0,0,-1,0],[9E+09,9E+09,9E+09,9E+09,9E+09,9E+09]];
    CONST robtarget T1827:=[[86.300026,129.593877,14.600035],[0.000000,0.000000,1.000000,0.000000],[0,0,-1,0],[9E+09,9E+09,9E+09,9E+09,9E+09,9E+09]];
    CONST robtarget T1828:=[[87.560031,129.413129,14.600035],[0.000000,0.000000,1.000000,0.000000],[0,0,-1,0],[9E+09,9E+09,9E+09,9E+09,9E+09,9E+09]];
    CONST robtarget T1829:=[[87.560031,83.409593,14.600035],[0.000000,0.000000,1.000000,0.000000],[0,0,-1,0],[9E+09,9E+09,9E+09,9E+09,9E+09,9E+09]];
    CONST robtarget T1830:=[[87.560031,76.590415,14.600035],[0.000000,0.000000,1.000000,0.000000],[0,0,-1,0],[9E+09,9E+09,9E+09,9E+09,9E+09,9E+09]];
    CONST robtarget T1831:=[[87.560031,30.586879,14.600035],[0.000000,0.000000,1.000000,0.000000],[0,0,-1,0],[9E+09,9E+09,9E+09,9E+09,9E+09,9E+09]];
    CONST robtarget T1832:=[[88.820035,30.786444,14.600035],[0.000000,0.000000,1.000000,0.000000],[0,0,-1,0],[9E+09,9E+09,9E+09,9E+09,9E+09,9E+09]];
    CONST robtarget T1833:=[[88.820035,129.213563,14.600035],[0.000000,0.000000,1.000000,0.000000],[0,0,-1,0],[9E+09,9E+09,9E+09,9E+09,9E+09,9E+09]];
    CONST robtarget T1834:=[[90.080040,128.960575,14.600035],[0.000000,0.000000,1.000000,0.000000],[0,0,-1,0],[9E+09,9E+09,9E+09,9E+09,9E+09,9E+09]];
    CONST robtarget T1835:=[[90.080040,31.039433,14.600035],[0.000000,0.000000,1.000000,0.000000],[0,0,-1,0],[9E+09,9E+09,9E+09,9E+09,9E+09,9E+09]];
    CONST robtarget T1836:=[[91.340044,31.307526,14.600035],[0.000000,0.000000,1.000000,0.000000],[0,0,-1,0],[9E+09,9E+09,9E+09,9E+09,9E+09,9E+09]];
    CONST robtarget T1837:=[[91.340044,128.692481,14.600035],[0.000000,0.000000,1.000000,0.000000],[0,0,-1,0],[9E+09,9E+09,9E+09,9E+09,9E+09,9E+09]];
    CONST robtarget T1838:=[[92.600049,128.374988,14.600035],[0.000000,0.000000,1.000000,0.000000],[0,0,-1,0],[9E+09,9E+09,9E+09,9E+09,9E+09,9E+09]];
    CONST robtarget T1839:=[[92.600049,31.625019,14.600035],[0.000000,0.000000,1.000000,0.000000],[0,0,-1,0],[9E+09,9E+09,9E+09,9E+09,9E+09,9E+09]];
    CONST robtarget T1840:=[[93.860053,31.969479,14.600035],[0.000000,0.000000,1.000000,0.000000],[0,0,-1,0],[9E+09,9E+09,9E+09,9E+09,9E+09,9E+09]];
    CONST robtarget T1841:=[[93.860053,128.030529,14.600035],[0.000000,0.000000,1.000000,0.000000],[0,0,-1,0],[9E+09,9E+09,9E+09,9E+09,9E+09,9E+09]];
    CONST robtarget T1842:=[[95.120058,127.652167,14.600035],[0.000000,0.000000,1.000000,0.000000],[0,0,-1,0],[9E+09,9E+09,9E+09,9E+09,9E+09,9E+09]];
    CONST robtarget T1843:=[[95.120058,32.347841,14.600035],[0.000000,0.000000,1.000000,0.000000],[0,0,-1,0],[9E+09,9E+09,9E+09,9E+09,9E+09,9E+09]];
    CONST robtarget T1844:=[[96.380062,32.772318,14.600035],[0.000000,0.000000,1.000000,0.000000],[0,0,-1,0],[9E+09,9E+09,9E+09,9E+09,9E+09,9E+09]];
    CONST robtarget T1845:=[[96.380062,127.227690,14.600035],[0.000000,0.000000,1.000000,0.000000],[0,0,-1,0],[9E+09,9E+09,9E+09,9E+09,9E+09,9E+09]];
    CONST robtarget T1846:=[[97.640067,126.783143,14.600035],[0.000000,0.000000,1.000000,0.000000],[0,0,-1,0],[9E+09,9E+09,9E+09,9E+09,9E+09,9E+09]];
    CONST robtarget T1847:=[[97.640067,33.216864,14.600035],[0.000000,0.000000,1.000000,0.000000],[0,0,-1,0],[9E+09,9E+09,9E+09,9E+09,9E+09,9E+09]];
    CONST robtarget T1848:=[[98.900071,33.722290,14.600035],[0.000000,0.000000,1.000000,0.000000],[0,0,-1,0],[9E+09,9E+09,9E+09,9E+09,9E+09,9E+09]];
    CONST robtarget T1849:=[[98.900071,126.277717,14.600035],[0.000000,0.000000,1.000000,0.000000],[0,0,-1,0],[9E+09,9E+09,9E+09,9E+09,9E+09,9E+09]];
    CONST robtarget T1850:=[[100.160076,125.745278,14.600035],[0.000000,0.000000,1.000000,0.000000],[0,0,-1,0],[9E+09,9E+09,9E+09,9E+09,9E+09,9E+09]];
    CONST robtarget T1851:=[[100.160076,34.254730,14.600035],[0.000000,0.000000,1.000000,0.000000],[0,0,-1,0],[9E+09,9E+09,9E+09,9E+09,9E+09,9E+09]];
    CONST robtarget T1852:=[[101.420080,34.827050,14.600035],[0.000000,0.000000,1.000000,0.000000],[0,0,-1,0],[9E+09,9E+09,9E+09,9E+09,9E+09,9E+09]];
    CONST robtarget T1853:=[[101.420080,125.172958,14.600035],[0.000000,0.000000,1.000000,0.000000],[0,0,-1,0],[9E+09,9E+09,9E+09,9E+09,9E+09,9E+09]];
    CONST robtarget T1854:=[[102.680085,124.546114,14.600035],[0.000000,0.000000,1.000000,0.000000],[0,0,-1,0],[9E+09,9E+09,9E+09,9E+09,9E+09,9E+09]];
    CONST robtarget T1855:=[[102.680085,35.453894,14.600035],[0.000000,0.000000,1.000000,0.000000],[0,0,-1,0],[9E+09,9E+09,9E+09,9E+09,9E+09,9E+09]];
    CONST robtarget T1856:=[[103.940089,36.110177,14.600035],[0.000000,0.000000,1.000000,0.000000],[0,0,-1,0],[9E+09,9E+09,9E+09,9E+09,9E+09,9E+09]];
    CONST robtarget T1857:=[[103.940089,123.889831,14.600035],[0.000000,0.000000,1.000000,0.000000],[0,0,-1,0],[9E+09,9E+09,9E+09,9E+09,9E+09,9E+09]];
    CONST robtarget T1858:=[[105.200094,123.174878,14.600035],[0.000000,0.000000,1.000000,0.000000],[0,0,-1,0],[9E+09,9E+09,9E+09,9E+09,9E+09,9E+09]];
    CONST robtarget T1859:=[[105.200094,36.825129,14.600035],[0.000000,0.000000,1.000000,0.000000],[0,0,-1,0],[9E+09,9E+09,9E+09,9E+09,9E+09,9E+09]];
    CONST robtarget T1860:=[[106.460098,37.589739,14.600035],[0.000000,0.000000,1.000000,0.000000],[0,0,-1,0],[9E+09,9E+09,9E+09,9E+09,9E+09,9E+09]];
    CONST robtarget T1861:=[[106.460098,122.410268,14.600035],[0.000000,0.000000,1.000000,0.000000],[0,0,-1,0],[9E+09,9E+09,9E+09,9E+09,9E+09,9E+09]];
    CONST robtarget T1862:=[[107.720103,121.607260,14.600035],[0.000000,0.000000,1.000000,0.000000],[0,0,-1,0],[9E+09,9E+09,9E+09,9E+09,9E+09,9E+09]];
    CONST robtarget T1863:=[[107.720103,81.789524,14.600035],[0.000000,0.000000,1.000000,0.000000],[0,0,-1,0],[9E+09,9E+09,9E+09,9E+09,9E+09,9E+09]];
    CONST robtarget T1864:=[[107.720103,78.210483,14.600035],[0.000000,0.000000,1.000000,0.000000],[0,0,-1,0],[9E+09,9E+09,9E+09,9E+09,9E+09,9E+09]];
    CONST robtarget T1865:=[[107.720103,38.392748,14.600035],[0.000000,0.000000,1.000000,0.000000],[0,0,-1,0],[9E+09,9E+09,9E+09,9E+09,9E+09,9E+09]];
    CONST robtarget T1866:=[[108.980107,39.265681,14.600035],[0.000000,0.000000,1.000000,0.000000],[0,0,-1,0],[9E+09,9E+09,9E+09,9E+09,9E+09,9E+09]];
    CONST robtarget T1867:=[[108.980107,75.547902,14.600035],[0.000000,0.000000,1.000000,0.000000],[0,0,-1,0],[9E+09,9E+09,9E+09,9E+09,9E+09,9E+09]];
    CONST robtarget T1868:=[[108.980107,84.452106,14.600035],[0.000000,0.000000,1.000000,0.000000],[0,0,-1,0],[9E+09,9E+09,9E+09,9E+09,9E+09,9E+09]];
    CONST robtarget T1869:=[[108.980107,120.734326,14.600035],[0.000000,0.000000,1.000000,0.000000],[0,0,-1,0],[9E+09,9E+09,9E+09,9E+09,9E+09,9E+09]];
    CONST robtarget T1870:=[[110.240112,119.803025,14.600035],[0.000000,0.000000,1.000000,0.000000],[0,0,-1,0],[9E+09,9E+09,9E+09,9E+09,9E+09,9E+09]];
    CONST robtarget T1871:=[[110.240112,85.779969,14.600035],[0.000000,0.000000,1.000000,0.000000],[0,0,-1,0],[9E+09,9E+09,9E+09,9E+09,9E+09,9E+09]];
    CONST robtarget T1872:=[[110.240112,74.220038,14.600035],[0.000000,0.000000,1.000000,0.000000],[0,0,-1,0],[9E+09,9E+09,9E+09,9E+09,9E+09,9E+09]];
    CONST robtarget T1873:=[[110.240112,40.196983,14.600035],[0.000000,0.000000,1.000000,0.000000],[0,0,-1,0],[9E+09,9E+09,9E+09,9E+09,9E+09,9E+09]];
    CONST robtarget T1874:=[[111.500116,41.180273,14.600035],[0.000000,0.000000,1.000000,0.000000],[0,0,-1,0],[9E+09,9E+09,9E+09,9E+09,9E+09,9E+09]];
    CONST robtarget T1875:=[[111.500116,73.379202,14.600035],[0.000000,0.000000,1.000000,0.000000],[0,0,-1,0],[9E+09,9E+09,9E+09,9E+09,9E+09,9E+09]];
    CONST robtarget T1876:=[[111.500116,86.620805,14.600035],[0.000000,0.000000,1.000000,0.000000],[0,0,-1,0],[9E+09,9E+09,9E+09,9E+09,9E+09,9E+09]];
    CONST robtarget T1877:=[[111.500116,118.819735,14.600035],[0.000000,0.000000,1.000000,0.000000],[0,0,-1,0],[9E+09,9E+09,9E+09,9E+09,9E+09,9E+09]];
    CONST robtarget T1878:=[[112.760121,117.767805,14.600035],[0.000000,0.000000,1.000000,0.000000],[0,0,-1,0],[9E+09,9E+09,9E+09,9E+09,9E+09,9E+09]];
    CONST robtarget T1879:=[[112.760121,87.152583,14.600035],[0.000000,0.000000,1.000000,0.000000],[0,0,-1,0],[9E+09,9E+09,9E+09,9E+09,9E+09,9E+09]];
    CONST robtarget T1880:=[[112.760121,72.847425,14.600035],[0.000000,0.000000,1.000000,0.000000],[0,0,-1,0],[9E+09,9E+09,9E+09,9E+09,9E+09,9E+09]];
    CONST robtarget T1881:=[[112.760121,42.232203,14.600035],[0.000000,0.000000,1.000000,0.000000],[0,0,-1,0],[9E+09,9E+09,9E+09,9E+09,9E+09,9E+09]];
    CONST robtarget T1882:=[[114.020125,43.373063,14.600035],[0.000000,0.000000,1.000000,0.000000],[0,0,-1,0],[9E+09,9E+09,9E+09,9E+09,9E+09,9E+09]];
    CONST robtarget T1883:=[[114.020125,72.576253,14.600035],[0.000000,0.000000,1.000000,0.000000],[0,0,-1,0],[9E+09,9E+09,9E+09,9E+09,9E+09,9E+09]];
    CONST robtarget T1884:=[[114.020125,87.423755,14.600035],[0.000000,0.000000,1.000000,0.000000],[0,0,-1,0],[9E+09,9E+09,9E+09,9E+09,9E+09,9E+09]];
    CONST robtarget T1885:=[[114.020125,116.626944,14.600035],[0.000000,0.000000,1.000000,0.000000],[0,0,-1,0],[9E+09,9E+09,9E+09,9E+09,9E+09,9E+09]];
    CONST robtarget T1886:=[[115.280130,115.412758,14.600035],[0.000000,0.000000,1.000000,0.000000],[0,0,-1,0],[9E+09,9E+09,9E+09,9E+09,9E+09,9E+09]];
    CONST robtarget T1887:=[[115.280130,87.487316,14.600035],[0.000000,0.000000,1.000000,0.000000],[0,0,-1,0],[9E+09,9E+09,9E+09,9E+09,9E+09,9E+09]];
    CONST robtarget T1888:=[[115.280130,72.512692,14.600035],[0.000000,0.000000,1.000000,0.000000],[0,0,-1,0],[9E+09,9E+09,9E+09,9E+09,9E+09,9E+09]];
    CONST robtarget T1889:=[[115.280130,44.587250,14.600035],[0.000000,0.000000,1.000000,0.000000],[0,0,-1,0],[9E+09,9E+09,9E+09,9E+09,9E+09,9E+09]];
    CONST robtarget T1890:=[[116.540134,45.884908,14.600035],[0.000000,0.000000,1.000000,0.000000],[0,0,-1,0],[9E+09,9E+09,9E+09,9E+09,9E+09,9E+09]];
    CONST robtarget T1891:=[[116.540134,72.670297,14.600035],[0.000000,0.000000,1.000000,0.000000],[0,0,-1,0],[9E+09,9E+09,9E+09,9E+09,9E+09,9E+09]];
    CONST robtarget T1892:=[[116.540134,87.329711,14.600035],[0.000000,0.000000,1.000000,0.000000],[0,0,-1,0],[9E+09,9E+09,9E+09,9E+09,9E+09,9E+09]];
    CONST robtarget T1893:=[[116.540134,114.115099,14.600035],[0.000000,0.000000,1.000000,0.000000],[0,0,-1,0],[9E+09,9E+09,9E+09,9E+09,9E+09,9E+09]];
    CONST robtarget T1894:=[[117.800139,112.721391,14.600035],[0.000000,0.000000,1.000000,0.000000],[0,0,-1,0],[9E+09,9E+09,9E+09,9E+09,9E+09,9E+09]];
    CONST robtarget T1895:=[[117.800139,86.948670,14.600035],[0.000000,0.000000,1.000000,0.000000],[0,0,-1,0],[9E+09,9E+09,9E+09,9E+09,9E+09,9E+09]];
    CONST robtarget T1896:=[[117.800139,73.051337,14.600035],[0.000000,0.000000,1.000000,0.000000],[0,0,-1,0],[9E+09,9E+09,9E+09,9E+09,9E+09,9E+09]];
    CONST robtarget T1897:=[[117.800139,47.278617,14.600035],[0.000000,0.000000,1.000000,0.000000],[0,0,-1,0],[9E+09,9E+09,9E+09,9E+09,9E+09,9E+09]];
    CONST robtarget T1898:=[[119.060143,48.787854,14.600035],[0.000000,0.000000,1.000000,0.000000],[0,0,-1,0],[9E+09,9E+09,9E+09,9E+09,9E+09,9E+09]];
    CONST robtarget T1899:=[[119.060143,73.708792,14.600035],[0.000000,0.000000,1.000000,0.000000],[0,0,-1,0],[9E+09,9E+09,9E+09,9E+09,9E+09,9E+09]];
    CONST robtarget T1900:=[[119.060143,86.291215,14.600035],[0.000000,0.000000,1.000000,0.000000],[0,0,-1,0],[9E+09,9E+09,9E+09,9E+09,9E+09,9E+09]];
    CONST robtarget T1901:=[[119.060143,111.212154,14.600035],[0.000000,0.000000,1.000000,0.000000],[0,0,-1,0],[9E+09,9E+09,9E+09,9E+09,9E+09,9E+09]];
    CONST robtarget T1902:=[[120.320148,109.560940,14.600035],[0.000000,0.000000,1.000000,0.000000],[0,0,-1,0],[9E+09,9E+09,9E+09,9E+09,9E+09,9E+09]];
    CONST robtarget T1903:=[[120.320148,85.271589,14.600035],[0.000000,0.000000,1.000000,0.000000],[0,0,-1,0],[9E+09,9E+09,9E+09,9E+09,9E+09,9E+09]];
    CONST robtarget T1904:=[[120.320148,74.728418,14.600035],[0.000000,0.000000,1.000000,0.000000],[0,0,-1,0],[9E+09,9E+09,9E+09,9E+09,9E+09,9E+09]];
    CONST robtarget T1905:=[[120.320148,50.439068,14.600035],[0.000000,0.000000,1.000000,0.000000],[0,0,-1,0],[9E+09,9E+09,9E+09,9E+09,9E+09,9E+09]];
    CONST robtarget T1906:=[[121.580152,52.240778,14.600035],[0.000000,0.000000,1.000000,0.000000],[0,0,-1,0],[9E+09,9E+09,9E+09,9E+09,9E+09,9E+09]];
    CONST robtarget T1907:=[[121.580152,76.422528,14.600035],[0.000000,0.000000,1.000000,0.000000],[0,0,-1,0],[9E+09,9E+09,9E+09,9E+09,9E+09,9E+09]];
    CONST robtarget T1908:=[[121.580152,83.577479,14.600035],[0.000000,0.000000,1.000000,0.000000],[0,0,-1,0],[9E+09,9E+09,9E+09,9E+09,9E+09,9E+09]];
    CONST robtarget T1909:=[[121.580152,107.759230,14.600035],[0.000000,0.000000,1.000000,0.000000],[0,0,-1,0],[9E+09,9E+09,9E+09,9E+09,9E+09,9E+09]];
    CONST robtarget T1910:=[[122.840157,105.775934,14.600035],[0.000000,0.000000,1.000000,0.000000],[0,0,-1,0],[9E+09,9E+09,9E+09,9E+09,9E+09,9E+09]];
    CONST robtarget T1911:=[[122.840157,54.224074,14.600035],[0.000000,0.000000,1.000000,0.000000],[0,0,-1,0],[9E+09,9E+09,9E+09,9E+09,9E+09,9E+09]];
    CONST robtarget T1912:=[[124.100161,56.444690,14.600035],[0.000000,0.000000,1.000000,0.000000],[0,0,-1,0],[9E+09,9E+09,9E+09,9E+09,9E+09,9E+09]];
    CONST robtarget T1913:=[[124.100161,103.555317,14.600035],[0.000000,0.000000,1.000000,0.000000],[0,0,-1,0],[9E+09,9E+09,9E+09,9E+09,9E+09,9E+09]];
    CONST robtarget T1914:=[[125.360166,101.007928,14.600035],[0.000000,0.000000,1.000000,0.000000],[0,0,-1,0],[9E+09,9E+09,9E+09,9E+09,9E+09,9E+09]];
    CONST robtarget T1915:=[[125.360166,58.992080,14.600035],[0.000000,0.000000,1.000000,0.000000],[0,0,-1,0],[9E+09,9E+09,9E+09,9E+09,9E+09,9E+09]];
    CONST robtarget T1916:=[[126.620170,61.953657,14.600035],[0.000000,0.000000,1.000000,0.000000],[0,0,-1,0],[9E+09,9E+09,9E+09,9E+09,9E+09,9E+09]];
    CONST robtarget T1917:=[[126.620170,98.046351,14.600035],[0.000000,0.000000,1.000000,0.000000],[0,0,-1,0],[9E+09,9E+09,9E+09,9E+09,9E+09,9E+09]];
    CONST robtarget T1918:=[[127.880175,94.360756,14.600035],[0.000000,0.000000,1.000000,0.000000],[0,0,-1,0],[9E+09,9E+09,9E+09,9E+09,9E+09,9E+09]];
    CONST robtarget T1919:=[[127.880175,65.639251,14.600035],[0.000000,0.000000,1.000000,0.000000],[0,0,-1,0],[9E+09,9E+09,9E+09,9E+09,9E+09,9E+09]];
    CONST robtarget T1920:=[[129.140179,70.797151,14.600035],[0.000000,0.000000,1.000000,0.000000],[0,0,-1,0],[9E+09,9E+09,9E+09,9E+09,9E+09,9E+09]];
    CONST robtarget T1921:=[[129.140179,89.202857,14.600035],[0.000000,0.000000,1.000000,0.000000],[0,0,-1,0],[9E+09,9E+09,9E+09,9E+09,9E+09,9E+09]];

PROC cladding()
    !Reset doLDLStartST;

